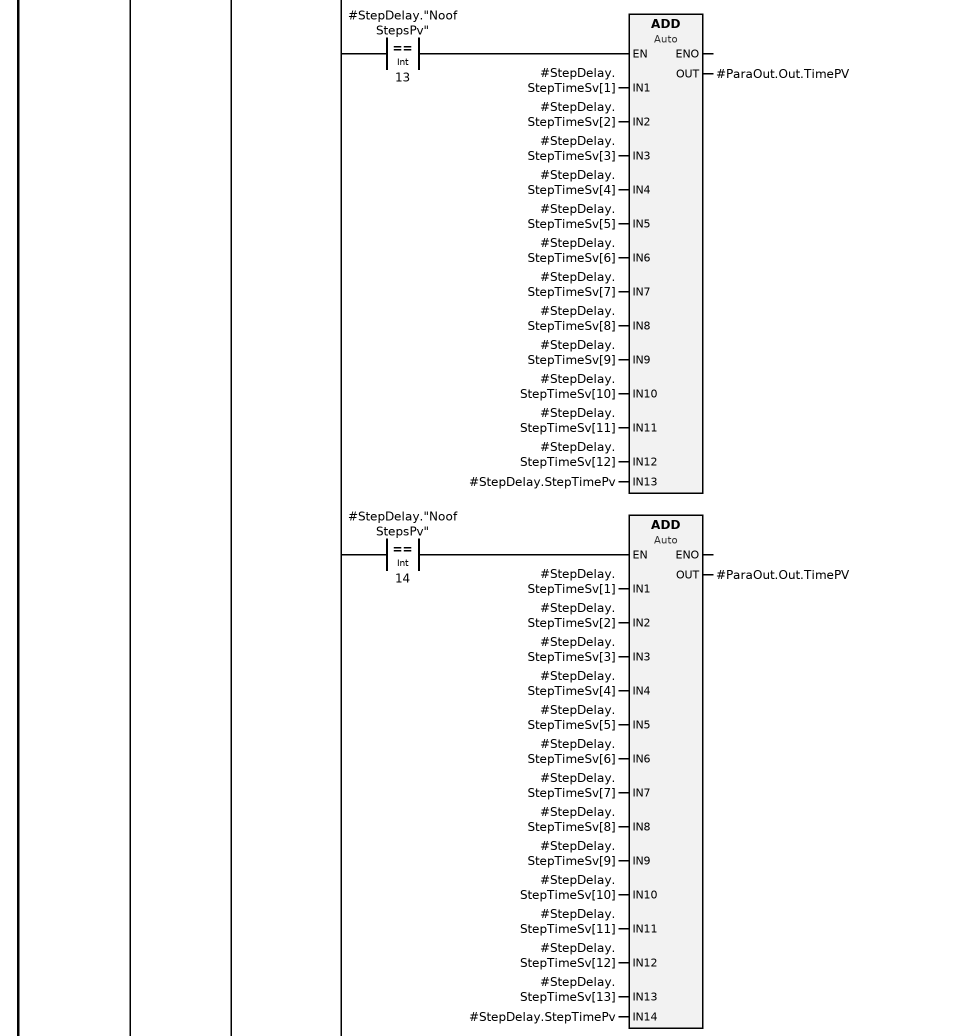
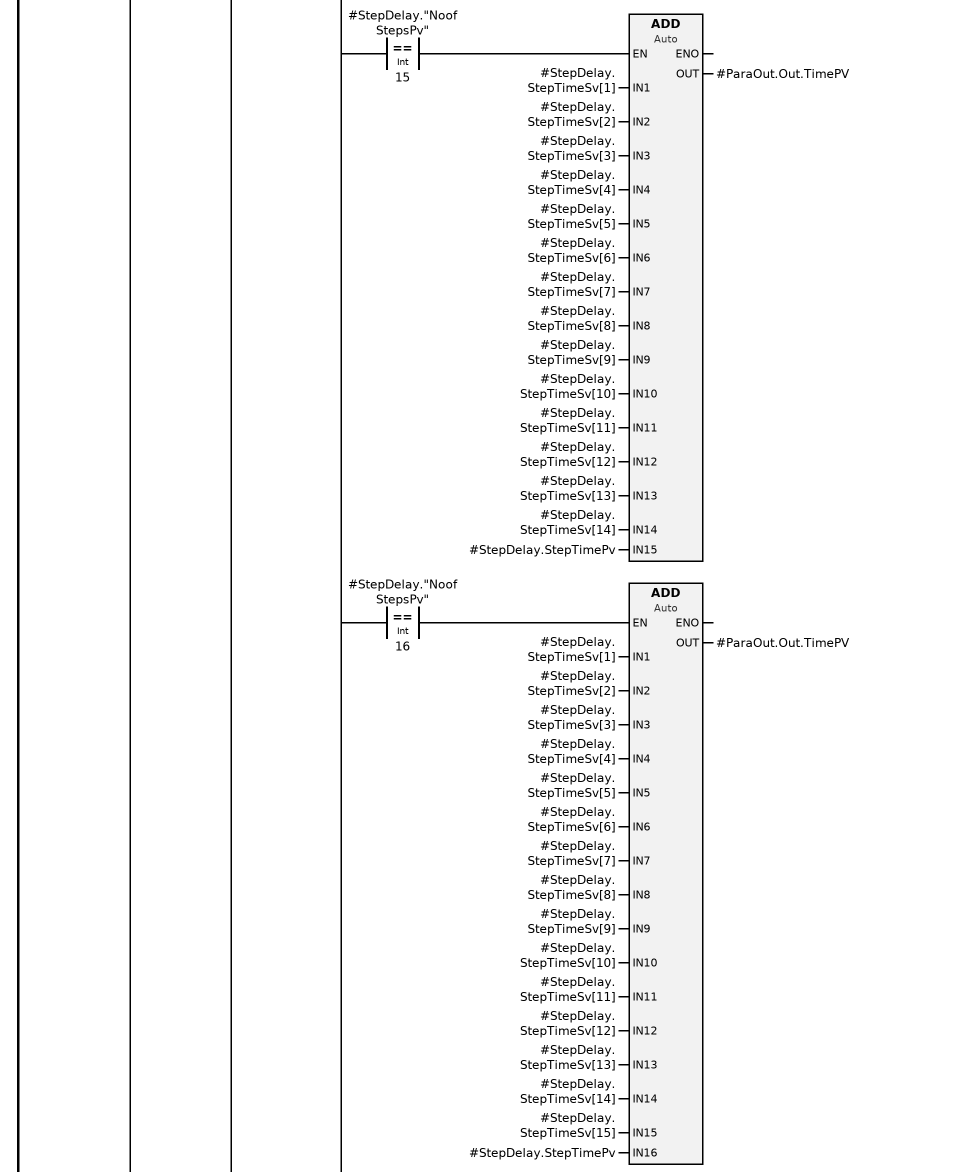
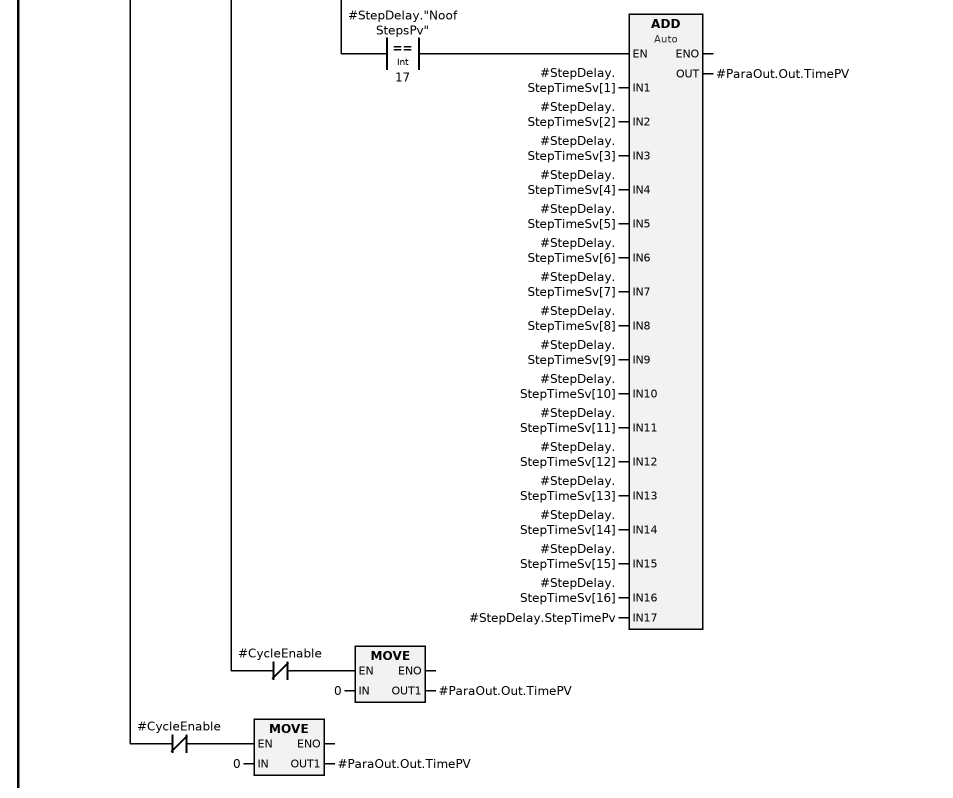
   RUNG wire#powerrail
      Contact( "AlwaysTRUE" )
      wire#w1
      { S7_Templates := "SrcType := DInt" } GE_Contact(in1 := #StepDelay.StepTimePv, in2 := 0)
      wire#w2
      { S7_Templates := "SrcType := Int" } LE_Contact(in1 := #ParaIn.PreciseEngineering.Loops, in2 := 20)
      wire#w3
      Add(in1 := #StepDelay.StepTimeSv[1], in2 := #StepDelay.StepTimeSv[2], in3 := #StepDelay.StepTimeSv[3], in4 := #StepDelay.StepTimeSv[4], in5 := #StepDelay.StepTimeSv[5], in6 := #StepDelay.StepTimeSv[6], in7 := #StepDelay.StepTimeSv[7], in8 := #StepDelay.StepTimeSv[8], in9 := #StepDelay.StepTimeSv[9], in10 := #StepDelay.StepTimeSv[10], in11 := #StepDelay.StepTimeSv[11], in12 := #StepDelay.StepTimeSv[12], in13 := #StepDelay.StepTimeSv[13], in14 := #StepDelay.StepTimeSv[14], in15 := #StepDelay.StepTimeSv[15], in16 := #StepDelay.StepTimeSv[16], in17 := #StepDelay.StepTimeSv[17], out => #ParaOut.Out.TimeSV)
   END_RUNG
   RUNG wire#w3
      Contact( #OverTemp )
      Add(in1 := #StepDelay.StepTimeSv[1], in2 := #StepDelay.StepTimeSv[2], in3 := #StepDelay.StepTimeSv[3], in4 := #StepDelay.StepTimeSv[4], in5 := #StepDelay.StepTimeSv[5], in6 := #StepDelay.StepTimeSv[6], in7 := #StepDelay.StepTimeSv[7], in8 := #StepDelay.StepTimeSv[8], in9 := #StepDelay.StepTimeSv[9], in10 := #StepDelay.StepTimeSv[10], in11 := #StepDelay.StepTimeSv[11], in12 := #StepDelay.StepTimeSv[12], in13 := #StepDelay.StepTimeSv[13], in14 := #StepDelay.StepTimeSv[14], in15 := #StepDelay.StepTimeSv[15], in16 := #StepDelay.StepTimeSv[16], in17 := #StepDelay.StepTimeSv[17], out => #ParaOut.Out.TimePV)
   END_RUNG
   RUNG wire#w2
      { S7_Templates := "SrcType := Int" } EQ_Contact(in1 := #ParaIn.PreciseEngineering.Loops, in2 := 5)
      I_Contact( #AlwaysTrue )
      wire#w4
      Add(in1 := #StepDelay.StepTimeSv[1], in2 := #StepDelay.StepTimeSv[2], in3 := #StepDelay.StepTimeSv[3], in4 := #StepDelay.StepTimeSv[4], in5 := #StepDelay.StepTimeSv[5], out => #ParaOut.Out.TimeSV)
   END_RUNG
   RUNG wire#w4
      Contact( #OverTemp )
      Add(in1 := #StepDelay.StepTimeSv[1], in2 := #StepDelay.StepTimeSv[2], in3 := #StepDelay.StepTimeSv[3], in4 := #StepDelay.StepTimeSv[4], in5 := #StepDelay.StepTimeSv[5], out => #ParaOut.Out.TimePV)
   END_RUNG
   RUNG wire#w2
      Contact( #CycleEnable )
      wire#w5
      { S7_Templates := "SrcType := Int" } EQ_Contact(in1 := #StepDelay."Noof StepsPv", in2 := 1)
      Move(in := #StepDelay.StepTimePv, out1 => #ParaOut.Out.TimePV)
   END_RUNG
   RUNG wire#w5
      { S7_Templates := "SrcType := Int" } EQ_Contact(in1 := #StepDelay."Noof StepsPv", in2 := 2)
      Add(in1 := #StepDelay.StepTimeSv[1], in2 := #StepDelay.StepTimePv, out => #ParaOut.Out.TimePV)
   END_RUNG
   RUNG wire#w5
      { S7_Templates := "SrcType := Int" } EQ_Contact(in1 := #StepDelay."Noof StepsPv", in2 := 3)
      Add(in1 := #StepDelay.StepTimeSv[1], in2 := #StepDelay.StepTimeSv[2], in3 := #StepDelay.StepTimePv, out => #ParaOut.Out.TimePV)
   END_RUNG
   RUNG wire#w5
      { S7_Templates := "SrcType := Int" } EQ_Contact(in1 := #StepDelay."Noof StepsPv", in2 := 4)
      Add(in1 := #StepDelay.StepTimeSv[1], in2 := #StepDelay.StepTimeSv[2], in3 := #StepDelay.StepTimeSv[3], in4 := #StepDelay.StepTimePv, out => #ParaOut.Out.TimePV)
   END_RUNG
   RUNG wire#w5
      { S7_Templates := "SrcType := Int" } EQ_Contact(in1 := #StepDelay."Noof StepsPv", in2 := 5)
      Add(in1 := #StepDelay.StepTimeSv[1], in2 := #StepDelay.StepTimeSv[2], in3 := #StepDelay.StepTimeSv[3], in4 := #StepDelay.StepTimeSv[4], in5 := #StepDelay.StepTimePv, out => #ParaOut.Out.TimePV)
   END_RUNG
   RUNG wire#w5
      { S7_Templates := "SrcType := Int" } EQ_Contact(in1 := #StepDelay."Noof StepsPv", in2 := 6)
      Add(in1 := #StepDelay.StepTimeSv[1], in2 := #StepDelay.StepTimeSv[2], in3 := #StepDelay.StepTimeSv[3], in4 := #StepDelay.StepTimeSv[4], in5 := #StepDelay.StepTimeSv[5], in6 := #StepDelay.StepTimePv, out => #ParaOut.Out.TimePV)
   END_RUNG
   RUNG wire#w5
      { S7_Templates := "SrcType := Int" } EQ_Contact(in1 := #StepDelay."Noof StepsPv", in2 := 7)
      Add(in1 := #StepDelay.StepTimeSv[1], in2 := #StepDelay.StepTimeSv[2], in3 := #StepDelay.StepTimeSv[3], in4 := #StepDelay.StepTimeSv[4], in5 := #StepDelay.StepTimeSv[5], in6 := #StepDelay.StepTimeSv[6], in7 := #StepDelay.StepTimePv, out => #ParaOut.Out.TimePV)
   END_RUNG
   RUNG wire#w5
      { S7_Templates := "SrcType := Int" } EQ_Contact(in1 := #StepDelay."Noof StepsPv", in2 := 8)
      Add(in1 := #StepDelay.StepTimeSv[1], in2 := #StepDelay.StepTimeSv[2], in3 := #StepDelay.StepTimeSv[3], in4 := #StepDelay.StepTimeSv[4], in5 := #StepDelay.StepTimeSv[5], in6 := #StepDelay.StepTimeSv[6], in7 := #StepDelay.StepTimeSv[7], in8 := #StepDelay.StepTimePv, out => #ParaOut.Out.TimePV)
   END_RUNG
   RUNG wire#w5
      { S7_Templates := "SrcType := Int" } EQ_Contact(in1 := #StepDelay."Noof StepsPv", in2 := 9)
      Add(in1 := #StepDelay.StepTimeSv[1], in2 := #StepDelay.StepTimeSv[2], in3 := #StepDelay.StepTimeSv[3], in4 := #StepDelay.StepTimeSv[4], in5 := #StepDelay.StepTimeSv[5], in6 := #StepDelay.StepTimeSv[6], in7 := #StepDelay.StepTimeSv[7], in8 := #StepDelay.StepTimeSv[8], in9 := #StepDelay.StepTimePv, out => #ParaOut.Out.TimePV)
   END_RUNG
   RUNG wire#w5
      { S7_Templates := "SrcType := Int" } EQ_Contact(in1 := #StepDelay."Noof StepsPv", in2 := 10)
      Add(in1 := #StepDelay.StepTimeSv[1], in2 := #StepDelay.StepTimeSv[2], in3 := #StepDelay.StepTimeSv[3], in4 := #StepDelay.StepTimeSv[4], in5 := #StepDelay.StepTimeSv[5], in6 := #StepDelay.StepTimeSv[6], in7 := #StepDelay.StepTimeSv[7], in8 := #StepDelay.StepTimeSv[8], in9 := #StepDelay.StepTimeSv[9], in10 := #StepDelay.StepTimePv, out => #ParaOut.Out.TimePV)
   END_RUNG
   RUNG wire#w5
      { S7_Templates := "SrcType := Int" } EQ_Contact(in1 := #StepDelay."Noof StepsPv", in2 := 11)
      Add(in1 := #StepDelay.StepTimeSv[1], in2 := #StepDelay.StepTimeSv[2], in3 := #StepDelay.StepTimeSv[3], in4 := #StepDelay.StepTimeSv[4], in5 := #StepDelay.StepTimeSv[5], in6 := #StepDelay.StepTimeSv[6], in7 := #StepDelay.StepTimeSv[7], in8 := #StepDelay.StepTimeSv[8], in9 := #StepDelay.StepTimeSv[9], in10 := #StepDelay.StepTimeSv[10], in11 := #StepDelay.StepTimePv, out => #ParaOut.Out.TimePV)
   END_RUNG
   RUNG wire#w5
      { S7_Templates := "SrcType := Int" } EQ_Contact(in1 := #StepDelay."Noof StepsPv", in2 := 12)
      Add(in1 := #StepDelay.StepTimeSv[1], in2 := #StepDelay.StepTimeSv[2], in3 := #StepDelay.StepTimeSv[3], in4 := #StepDelay.StepTimeSv[4], in5 := #StepDelay.StepTimeSv[5], in6 := #StepDelay.StepTimeSv[6], in7 := #StepDelay.StepTimeSv[7], in8 := #StepDelay.StepTimeSv[8], in9 := #StepDelay.StepTimeSv[9], in10 := #StepDelay.StepTimeSv[10], in11 := #StepDelay.StepTimeSv[11], in12 := #StepDelay.StepTimePv, out => #ParaOut.Out.TimePV)
   END_RUNG
   RUNG wire#w5
      { S7_Templates := "SrcType := Int" } EQ_Contact(in1 := #StepDelay."Noof StepsPv", in2 := 13)
      Add(in1 := #StepDelay.StepTimeSv[1], in2 := #StepDelay.StepTimeSv[2], in3 := #StepDelay.StepTimeSv[3], in4 := #StepDelay.StepTimeSv[4], in5 := #StepDelay.StepTimeSv[5], in6 := #StepDelay.StepTimeSv[6], in7 := #StepDelay.StepTimeSv[7], in8 := #StepDelay.StepTimeSv[8], in9 := #StepDelay.StepTimeSv[9], in10 := #StepDelay.StepTimeSv[10], in11 := #StepDelay.StepTimeSv[11], in12 := #StepDelay.StepTimeSv[12], in13 := #StepDelay.StepTimePv, out => #ParaOut.Out.TimePV)
   END_RUNG
   RUNG wire#w5
      { S7_Templates := "SrcType := Int" } EQ_Contact(in1 := #StepDelay."Noof StepsPv", in2 := 14)
      Add(in1 := #StepDelay.StepTimeSv[1], in2 := #StepDelay.StepTimeSv[2], in3 := #StepDelay.StepTimeSv[3], in4 := #StepDelay.StepTimeSv[4], in5 := #StepDelay.StepTimeSv[5], in6 := #StepDelay.StepTimeSv[6], in7 := #StepDelay.StepTimeSv[7], in8 := #StepDelay.StepTimeSv[8], in9 := #StepDelay.StepTimeSv[9], in10 := #StepDelay.StepTimeSv[10], in11 := #StepDelay.StepTimeSv[11], in12 := #StepDelay.StepTimeSv[12], in13 := #StepDelay.StepTimeSv[13], in14 := #StepDelay.StepTimePv, out => #ParaOut.Out.TimePV)
   END_RUNG
   RUNG wire#w5
      { S7_Templates := "SrcType := Int" } EQ_Contact(in1 := #StepDelay."Noof StepsPv", in2 := 15)
      Add(in1 := #StepDelay.StepTimeSv[1], in2 := #StepDelay.StepTimeSv[2], in3 := #StepDelay.StepTimeSv[3], in4 := #StepDelay.StepTimeSv[4], in5 := #StepDelay.StepTimeSv[5], in6 := #StepDelay.StepTimeSv[6], in7 := #StepDelay.StepTimeSv[7], in8 := #StepDelay.StepTimeSv[8], in9 := #StepDelay.StepTimeSv[9], in10 := #StepDelay.StepTimeSv[10], in11 := #StepDelay.StepTimeSv[11], in12 := #StepDelay.StepTimeSv[12], in13 := #StepDelay.StepTimeSv[13], in14 := #StepDelay.StepTimeSv[14], in15 := #StepDelay.StepTimePv, out => #ParaOut.Out.TimePV)
   END_RUNG
   RUNG wire#w5
      { S7_Templates := "SrcType := Int" } EQ_Contact(in1 := #StepDelay."Noof StepsPv", in2 := 16)
      Add(in1 := #StepDelay.StepTimeSv[1], in2 := #StepDelay.StepTimeSv[2], in3 := #StepDelay.StepTimeSv[3], in4 := #StepDelay.StepTimeSv[4], in5 := #StepDelay.StepTimeSv[5], in6 := #StepDelay.StepTimeSv[6], in7 := #StepDelay.StepTimeSv[7], in8 := #StepDelay.StepTimeSv[8], in9 := #StepDelay.StepTimeSv[9], in10 := #StepDelay.StepTimeSv[10], in11 := #StepDelay.StepTimeSv[11], in12 := #StepDelay.StepTimeSv[12], in13 := #StepDelay.StepTimeSv[13], in14 := #StepDelay.StepTimeSv[14], in15 := #StepDelay.StepTimeSv[15], in16 := #StepDelay.StepTimePv, out => #ParaOut.Out.TimePV)
   END_RUNG
   RUNG wire#w5
      { S7_Templates := "SrcType := Int" } EQ_Contact(in1 := #StepDelay."Noof StepsPv", in2 := 17)
      Add(in1 := #StepDelay.StepTimeSv[1], in2 := #StepDelay.StepTimeSv[2], in3 := #StepDelay.StepTimeSv[3], in4 := #StepDelay.StepTimeSv[4], in5 := #StepDelay.StepTimeSv[5], in6 := #StepDelay.StepTimeSv[6], in7 := #StepDelay.StepTimeSv[7], in8 := #StepDelay.StepTimeSv[8], in9 := #StepDelay.StepTimeSv[9], in10 := #StepDelay.StepTimeSv[10], in11 := #StepDelay.StepTimeSv[11], in12 := #StepDelay.StepTimeSv[12], in13 := #StepDelay.StepTimeSv[13], in14 := #StepDelay.StepTimeSv[14], in15 := #StepDelay.StepTimeSv[15], in16 := #StepDelay.StepTimeSv[16], in17 := #StepDelay.StepTimePv, out => #ParaOut.Out.TimePV)
   END_RUNG
   RUNG wire#w2
      I_Contact( #CycleEnable )
      Move(in := 0, out1 => #ParaOut.Out.TimePV)
   END_RUNG
   RUNG wire#w1
      I_Contact( #CycleEnable )
      Move(in := 0, out1 => #ParaOut.Out.TimePV)
   END_RUNG
   // the same network as SCL:
   #_w1 := "AlwaysTRUE" AND (#StepDelay.StepTimePv >= 0);
   #_w2 := #_w1 AND (#ParaIn.PreciseEngineering.Loops <= 20);
   IF #_w2 THEN
       #ParaOut.Out.TimeSV := #StepDelay.StepTimeSv[1] + #StepDelay.StepTimeSv[2] + #StepDelay.StepTimeSv[3] + #StepDelay.StepTimeSv[4] + #StepDelay.StepTimeSv[5] + #StepDelay.StepTimeSv[6] + #StepDelay.StepTimeSv[7] + #StepDelay.StepTimeSv[8] + #StepDelay.StepTimeSv[9] + #StepDelay.StepTimeSv[10] + #StepDelay.StepTimeSv[11] + #StepDelay.StepTimeSv[12] + #StepDelay.StepTimeSv[13] + #StepDelay.StepTimeSv[14] + #StepDelay.StepTimeSv[15] + #StepDelay.StepTimeSv[16] + #StepDelay.StepTimeSv[17];
   END_IF;
   IF #_w2 AND #OverTemp THEN
       #ParaOut.Out.TimePV := #StepDelay.StepTimeSv[1] + #StepDelay.StepTimeSv[2] + #StepDelay.StepTimeSv[3] + #StepDelay.StepTimeSv[4] + #StepDelay.StepTimeSv[5] + #StepDelay.StepTimeSv[6] + #StepDelay.StepTimeSv[7] + #StepDelay.StepTimeSv[8] + #StepDelay.StepTimeSv[9] + #StepDelay.StepTimeSv[10] + #StepDelay.StepTimeSv[11] + #StepDelay.StepTimeSv[12] + #StepDelay.StepTimeSv[13] + #StepDelay.StepTimeSv[14] + #StepDelay.StepTimeSv[15] + #StepDelay.StepTimeSv[16] + #StepDelay.StepTimeSv[17];
   END_IF;
   #_w3 := #_w1 AND (#ParaIn.PreciseEngineering.Loops = 5) AND NOT #AlwaysTrue;
   IF #_w3 THEN
       #ParaOut.Out.TimeSV := #StepDelay.StepTimeSv[1] + #StepDelay.StepTimeSv[2] + #StepDelay.StepTimeSv[3] + #StepDelay.StepTimeSv[4] + #StepDelay.StepTimeSv[5];
   END_IF;
   IF #_w3 AND #OverTemp THEN
       #ParaOut.Out.TimePV := #StepDelay.StepTimeSv[1] + #StepDelay.StepTimeSv[2] + #StepDelay.StepTimeSv[3] + #StepDelay.StepTimeSv[4] + #StepDelay.StepTimeSv[5];
   END_IF;
   #_w4 := #_w1 AND #CycleEnable;
   IF #_w4 AND (#StepDelay."Noof StepsPv" = 1) THEN #ParaOut.Out.TimePV := #StepDelay.StepTimePv; END_IF;
   IF #_w4 AND (#StepDelay."Noof StepsPv" = 2) THEN
       #ParaOut.Out.TimePV := #StepDelay.StepTimeSv[1] + #StepDelay.StepTimePv;
   END_IF;
   IF #_w4 AND (#StepDelay."Noof StepsPv" = 3) THEN
       #ParaOut.Out.TimePV := #StepDelay.StepTimeSv[1] + #StepDelay.StepTimeSv[2] + #StepDelay.StepTimePv;
   END_IF;
   IF #_w4 AND (#StepDelay."Noof StepsPv" = 4) THEN
       #ParaOut.Out.TimePV := #StepDelay.StepTimeSv[1] + #StepDelay.StepTimeSv[2] + #StepDelay.StepTimeSv[3] + #StepDelay.StepTimePv;
   END_IF;
   IF #_w4 AND (#StepDelay."Noof StepsPv" = 5) THEN
       #ParaOut.Out.TimePV := #StepDelay.StepTimeSv[1] + #StepDelay.StepTimeSv[2] + #StepDelay.StepTimeSv[3] + #StepDelay.StepTimeSv[4] + #StepDelay.StepTimePv;
   END_IF;
   IF #_w4 AND (#StepDelay."Noof StepsPv" = 6) THEN
       #ParaOut.Out.TimePV := #StepDelay.StepTimeSv[1] + #StepDelay.StepTimeSv[2] + #StepDelay.StepTimeSv[3] + #StepDelay.StepTimeSv[4] + #StepDelay.StepTimeSv[5] + #StepDelay.StepTimePv;
   END_IF;
   IF #_w4 AND (#StepDelay."Noof StepsPv" = 7) THEN
       #ParaOut.Out.TimePV := #StepDelay.StepTimeSv[1] + #StepDelay.StepTimeSv[2] + #StepDelay.StepTimeSv[3] + #StepDelay.StepTimeSv[4] + #StepDelay.StepTimeSv[5] + #StepDelay.StepTimeSv[6] + #StepDelay.StepTimePv;
   END_IF;
   IF #_w4 AND (#StepDelay."Noof StepsPv" = 8) THEN
       #ParaOut.Out.TimePV := #StepDelay.StepTimeSv[1] + #StepDelay.StepTimeSv[2] + #StepDelay.StepTimeSv[3] + #StepDelay.StepTimeSv[4] + #StepDelay.StepTimeSv[5] + #StepDelay.StepTimeSv[6] + #StepDelay.StepTimeSv[7] + #StepDelay.StepTimePv;
   END_IF;
   IF #_w4 AND (#StepDelay."Noof StepsPv" = 9) THEN
       #ParaOut.Out.TimePV := #StepDelay.StepTimeSv[1] + #StepDelay.StepTimeSv[2] + #StepDelay.StepTimeSv[3] + #StepDelay.StepTimeSv[4] + #StepDelay.StepTimeSv[5] + #StepDelay.StepTimeSv[6] + #StepDelay.StepTimeSv[7] + #StepDelay.StepTimeSv[8] + #StepDelay.StepTimePv;
   END_IF;
   IF #_w4 AND (#StepDelay."Noof StepsPv" = 10) THEN
       #ParaOut.Out.TimePV := #StepDelay.StepTimeSv[1] + #StepDelay.StepTimeSv[2] + #StepDelay.StepTimeSv[3] + #StepDelay.StepTimeSv[4] + #StepDelay.StepTimeSv[5] + #StepDelay.StepTimeSv[6] + #StepDelay.StepTimeSv[7] + #StepDelay.StepTimeSv[8] + #StepDelay.StepTimeSv[9] + #StepDelay.StepTimePv;
   END_IF;
   IF #_w4 AND (#StepDelay."Noof StepsPv" = 11) THEN
       #ParaOut.Out.TimePV := #StepDelay.StepTimeSv[1] + #StepDelay.StepTimeSv[2] + #StepDelay.StepTimeSv[3] + #StepDelay.StepTimeSv[4] + #StepDelay.StepTimeSv[5] + #StepDelay.StepTimeSv[6] + #StepDelay.StepTimeSv[7] + #StepDelay.StepTimeSv[8] + #StepDelay.StepTimeSv[9] + #StepDelay.StepTimeSv[10] + #StepDelay.StepTimePv;
   END_IF;
   IF #_w4 AND (#StepDelay."Noof StepsPv" = 12) THEN
       #ParaOut.Out.TimePV := #StepDelay.StepTimeSv[1] + #StepDelay.StepTimeSv[2] + #StepDelay.StepTimeSv[3] + #StepDelay.StepTimeSv[4] + #StepDelay.StepTimeSv[5] + #StepDelay.StepTimeSv[6] + #StepDelay.StepTimeSv[7] + #StepDelay.StepTimeSv[8] + #StepDelay.StepTimeSv[9] + #StepDelay.StepTimeSv[10] + #StepDelay.StepTimeSv[11] + #StepDelay.StepTimePv;
   END_IF;
   IF #_w4 AND (#StepDelay."Noof StepsPv" = 13) THEN
       #ParaOut.Out.TimePV := #StepDelay.StepTimeSv[1] + #StepDelay.StepTimeSv[2] + #StepDelay.StepTimeSv[3] + #StepDelay.StepTimeSv[4] + #StepDelay.StepTimeSv[5] + #StepDelay.StepTimeSv[6] + #StepDelay.StepTimeSv[7] + #StepDelay.StepTimeSv[8] + #StepDelay.StepTimeSv[9] + #StepDelay.StepTimeSv[10] + #StepDelay.StepTimeSv[11] + #StepDelay.StepTimeSv[12] + #StepDelay.StepTimePv;
   END_IF;
   IF #_w4 AND (#StepDelay."Noof StepsPv" = 14) THEN
       #ParaOut.Out.TimePV := #StepDelay.StepTimeSv[1] + #StepDelay.StepTimeSv[2] + #StepDelay.StepTimeSv[3] + #StepDelay.StepTimeSv[4] + #StepDelay.StepTimeSv[5] + #StepDelay.StepTimeSv[6] + #StepDelay.StepTimeSv[7] + #StepDelay.StepTimeSv[8] + #StepDelay.StepTimeSv[9] + #StepDelay.StepTimeSv[10] + #StepDelay.StepTimeSv[11] + #StepDelay.StepTimeSv[12] + #StepDelay.StepTimeSv[13] + #StepDelay.StepTimePv;
   END_IF;
   IF #_w4 AND (#StepDelay."Noof StepsPv" = 15) THEN
       #ParaOut.Out.TimePV := #StepDelay.StepTimeSv[1] + #StepDelay.StepTimeSv[2] + #StepDelay.StepTimeSv[3] + #StepDelay.StepTimeSv[4] + #StepDelay.StepTimeSv[5] + #StepDelay.StepTimeSv[6] + #StepDelay.StepTimeSv[7] + #StepDelay.StepTimeSv[8] + #StepDelay.StepTimeSv[9] + #StepDelay.StepTimeSv[10] + #StepDelay.StepTimeSv[11] + #StepDelay.StepTimeSv[12] + #StepDelay.StepTimeSv[13] + #StepDelay.StepTimeSv[14] + #StepDelay.StepTimePv;
   END_IF;
   IF #_w4 AND (#StepDelay."Noof StepsPv" = 16) THEN
       #ParaOut.Out.TimePV := #StepDelay.StepTimeSv[1] + #StepDelay.StepTimeSv[2] + #StepDelay.StepTimeSv[3] + #StepDelay.StepTimeSv[4] + #StepDelay.StepTimeSv[5] + #StepDelay.StepTimeSv[6] + #StepDelay.StepTimeSv[7] + #StepDelay.StepTimeSv[8] + #StepDelay.StepTimeSv[9] + #StepDelay.StepTimeSv[10] + #StepDelay.StepTimeSv[11] + #StepDelay.StepTimeSv[12] + #StepDelay.StepTimeSv[13] + #StepDelay.StepTimeSv[14] + #StepDelay.StepTimeSv[15] + #StepDelay.StepTimePv;
   END_IF;
   IF #_w4 AND (#StepDelay."Noof StepsPv" = 17) THEN
       #ParaOut.Out.TimePV := #StepDelay.StepTimeSv[1] + #StepDelay.StepTimeSv[2] + #StepDelay.StepTimeSv[3] + #StepDelay.StepTimeSv[4] + #StepDelay.StepTimeSv[5] + #StepDelay.StepTimeSv[6] + #StepDelay.StepTimeSv[7] + #StepDelay.StepTimeSv[8] + #StepDelay.StepTimeSv[9] + #StepDelay.StepTimeSv[10] + #StepDelay.StepTimeSv[11] + #StepDelay.StepTimeSv[12] + #StepDelay.StepTimeSv[13] + #StepDelay.StepTimeSv[14] + #StepDelay.StepTimeSv[15] + #StepDelay.StepTimeSv[16] + #StepDelay.StepTimePv;
   END_IF;
   IF #_w1 AND NOT #CycleEnable THEN #ParaOut.Out.TimePV := 0; END_IF;
   IF "AlwaysTRUE" AND NOT #CycleEnable THEN #ParaOut.Out.TimePV := 0; END_IF;
END_REGION

REGION Network 12: #StepDelay
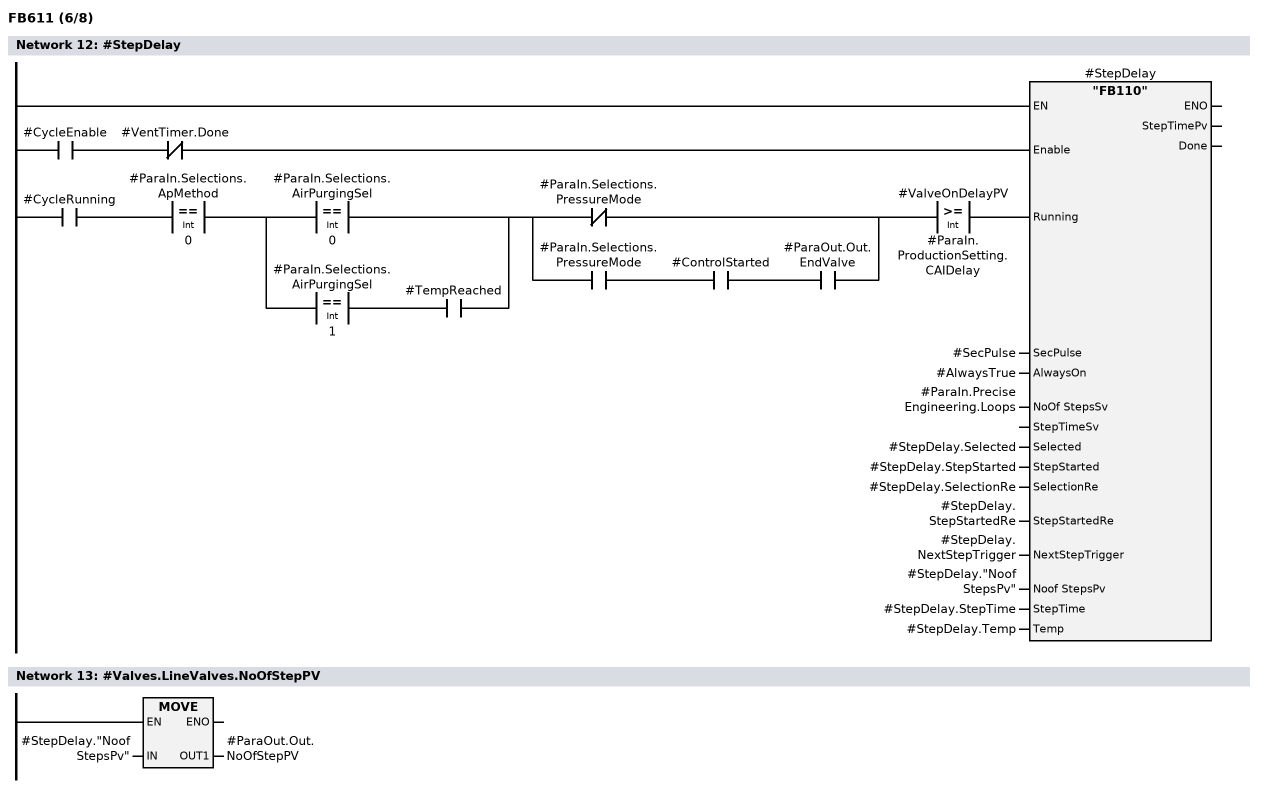
   RUNG wire#powerrail
      #StepDelay(Enable := wire#w1, Running := wire#w5, SecPulse := #SecPulse, AlwaysOn := #AlwaysTrue, "NoOf StepsSv" := #ParaIn.PreciseEngineering.Loops, StepTimeSv :=, Selected := #StepDelay.Selected, StepStarted := #StepDelay.StepStarted, SelectionRe := #StepDelay.SelectionRe, StepStartedRe := #StepDelay.StepStartedRe, NextStepTrigger := #StepDelay.NextStepTrigger, "Noof StepsPv" := #StepDelay."Noof StepsPv", StepTime := #StepDelay.StepTime, Temp := #StepDelay.Temp, StepTimePv =>, Done =>)
   END_RUNG
   RUNG wire#powerrail
      Contact( #CycleEnable )
      I_Contact( #VentTimer.Done )
   END_RUNG wire#w1
   RUNG wire#powerrail
      Contact( #CycleRunning )
      { S7_Templates := "SrcType := Int" } EQ_Contact(in1 := #ParaIn.Selections.ApMethod, in2 := 0)
      wire#w2
      { S7_Templates := "SrcType := Int" } EQ_Contact(in1 := #ParaIn.Selections.AirPurgingSel, in2 := 0)
      wire#w3
      I_Contact( #ParaIn.Selections.PressureMode )
      wire#w4
      { S7_Templates := "SrcType := Int" } GE_Contact(in1 := #ValveOnDelayPV, in2 := #ParaIn.ProductionSetting.CAIDelay)
   END_RUNG wire#w5
   RUNG wire#w2
      { S7_Templates := "SrcType := Int" } EQ_Contact(in1 := #ParaIn.Selections.AirPurgingSel, in2 := 1)
      Contact( #TempReached )
   END_RUNG wire#w3
   RUNG wire#w3
      Contact( #ParaIn.Selections.PressureMode )
      Contact( #ControlStarted )
      Contact( #ParaOut.Out.EndValve )
   END_RUNG wire#w4
   // the same network as SCL:
   #StepDelay(Enable := #CycleEnable AND NOT #VentTimer.Done,   // "FB110"
              Running := #CycleRunning AND (#ParaIn.Selections.ApMethod = 0) AND ((#ParaIn.Selections.AirPurgingSel = 0) OR ((#ParaIn.Selections.AirPurgingSel = 1) AND #TempReached)) AND (NOT #ParaIn.Selections.PressureMode OR (#ParaIn.Selections.PressureMode AND #ControlStarted AND #ParaOut.Out.EndValve)) AND (#ValveOnDelayPV >= #ParaIn.ProductionSetting.CAIDelay),
              SecPulse := #SecPulse,
              AlwaysOn := #AlwaysTrue,
              "NoOf StepsSv" := #ParaIn.PreciseEngineering.Loops,
              Selected := #StepDelay.Selected,
              StepStarted := #StepDelay.StepStarted,
              SelectionRe := #StepDelay.SelectionRe,
              StepStartedRe := #StepDelay.StepStartedRe,
              NextStepTrigger := #StepDelay.NextStepTrigger,
              "Noof StepsPv" := #StepDelay."Noof StepsPv",
              StepTime := #StepDelay.StepTime,
              Temp := #StepDelay.Temp);
END_REGION

REGION Network 13: #Valves.LineValves.NoOfStepPV
   RUNG wire#powerrail
      Move(in := #StepDelay."Noof StepsPv", out1 => #ParaOut.Out.NoOfStepPV)
   END_RUNG
   // the same network as SCL:
   #ParaOut.Out.NoOfStepPV := #StepDelay."Noof StepsPv";
END_REGION

REGION Network 14: Loop Outputs
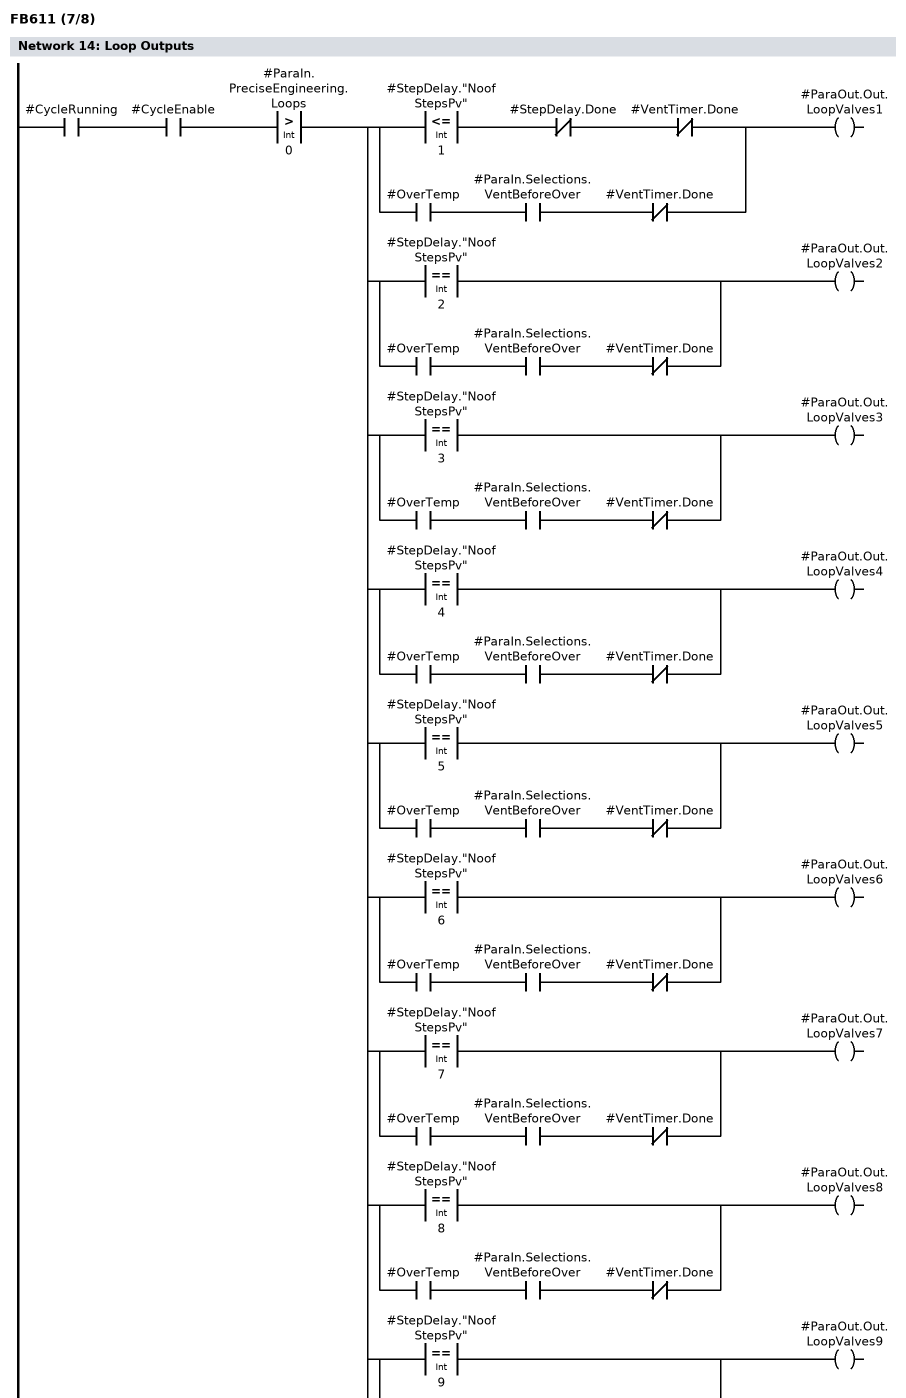
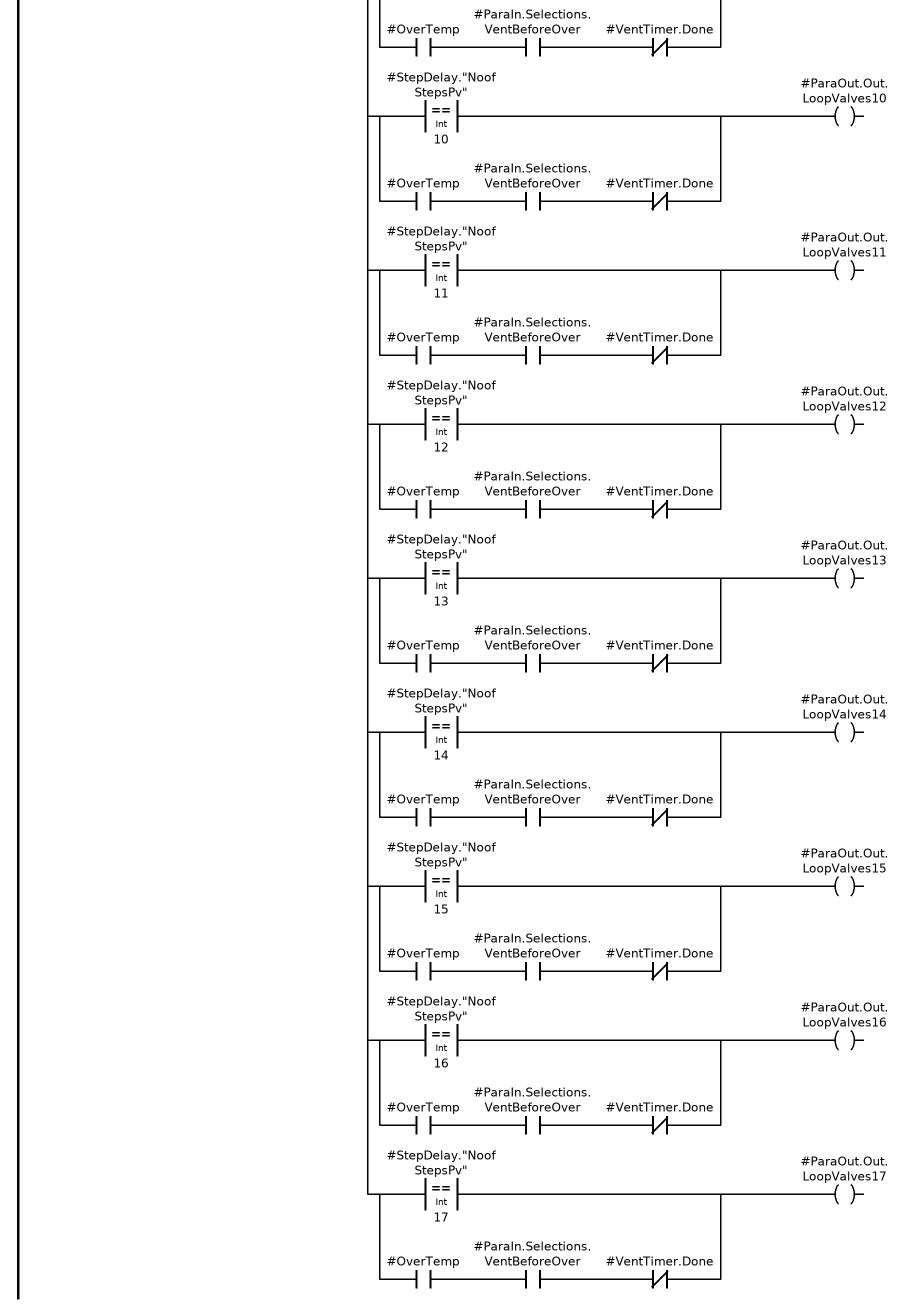
   RUNG wire#powerrail
      Contact( #CycleRunning )
      Contact( #CycleEnable )
      { S7_Templates := "SrcType := Int" } GT_Contact(in1 := #ParaIn.PreciseEngineering.Loops, in2 := 0)
      wire#w1
      { S7_Templates := "SrcType := Int" } LE_Contact(in1 := #StepDelay."Noof StepsPv", in2 := 1)
      I_Contact( #StepDelay.Done )
      I_Contact( #VentTimer.Done )
      wire#w2
      Coil( #ParaOut.Out.LoopValves1 )
   END_RUNG
   RUNG wire#w1
      Contact( #OverTemp )
      Contact( #ParaIn.Selections.VentBeforeOver )
      I_Contact( #VentTimer.Done )
   END_RUNG wire#w2
   RUNG wire#w1
      { S7_Templates := "SrcType := Int" } EQ_Contact(in1 := #StepDelay."Noof StepsPv", in2 := 2)
      wire#w3
      Coil( #ParaOut.Out.LoopValves2 )
   END_RUNG
   RUNG wire#w1
      Contact( #OverTemp )
      Contact( #ParaIn.Selections.VentBeforeOver )
      I_Contact( #VentTimer.Done )
   END_RUNG wire#w3
   RUNG wire#w1
      { S7_Templates := "SrcType := Int" } EQ_Contact(in1 := #StepDelay."Noof StepsPv", in2 := 3)
      wire#w4
      Coil( #ParaOut.Out.LoopValves3 )
   END_RUNG
   RUNG wire#w1
      Contact( #OverTemp )
      Contact( #ParaIn.Selections.VentBeforeOver )
      I_Contact( #VentTimer.Done )
   END_RUNG wire#w4
   RUNG wire#w1
      { S7_Templates := "SrcType := Int" } EQ_Contact(in1 := #StepDelay."Noof StepsPv", in2 := 4)
      wire#w5
      Coil( #ParaOut.Out.LoopValves4 )
   END_RUNG
   RUNG wire#w1
      Contact( #OverTemp )
      Contact( #ParaIn.Selections.VentBeforeOver )
      I_Contact( #VentTimer.Done )
   END_RUNG wire#w5
   RUNG wire#w1
      { S7_Templates := "SrcType := Int" } EQ_Contact(in1 := #StepDelay."Noof StepsPv", in2 := 5)
      wire#w6
      Coil( #ParaOut.Out.LoopValves5 )
   END_RUNG
   RUNG wire#w1
      Contact( #OverTemp )
      Contact( #ParaIn.Selections.VentBeforeOver )
      I_Contact( #VentTimer.Done )
   END_RUNG wire#w6
   RUNG wire#w1
      { S7_Templates := "SrcType := Int" } EQ_Contact(in1 := #StepDelay."Noof StepsPv", in2 := 6)
      wire#w7
      Coil( #ParaOut.Out.LoopValves6 )
   END_RUNG
   RUNG wire#w1
      Contact( #OverTemp )
      Contact( #ParaIn.Selections.VentBeforeOver )
      I_Contact( #VentTimer.Done )
   END_RUNG wire#w7
   RUNG wire#w1
      { S7_Templates := "SrcType := Int" } EQ_Contact(in1 := #StepDelay."Noof StepsPv", in2 := 7)
      wire#w8
      Coil( #ParaOut.Out.LoopValves7 )
   END_RUNG
   RUNG wire#w1
      Contact( #OverTemp )
      Contact( #ParaIn.Selections.VentBeforeOver )
      I_Contact( #VentTimer.Done )
   END_RUNG wire#w8
   RUNG wire#w1
      { S7_Templates := "SrcType := Int" } EQ_Contact(in1 := #StepDelay."Noof StepsPv", in2 := 8)
      wire#w9
      Coil( #ParaOut.Out.LoopValves8 )
   END_RUNG
   RUNG wire#w1
      Contact( #OverTemp )
      Contact( #ParaIn.Selections.VentBeforeOver )
      I_Contact( #VentTimer.Done )
   END_RUNG wire#w9
   RUNG wire#w1
      { S7_Templates := "SrcType := Int" } EQ_Contact(in1 := #StepDelay."Noof StepsPv", in2 := 9)
      wire#w10
      Coil( #ParaOut.Out.LoopValves9 )
   END_RUNG
   RUNG wire#w1
      Contact( #OverTemp )
      Contact( #ParaIn.Selections.VentBeforeOver )
      I_Contact( #VentTimer.Done )
   END_RUNG wire#w10
   RUNG wire#w1
      { S7_Templates := "SrcType := Int" } EQ_Contact(in1 := #StepDelay."Noof StepsPv", in2 := 10)
      wire#w11
      Coil( #ParaOut.Out.LoopValves10 )
   END_RUNG
   RUNG wire#w1
      Contact( #OverTemp )
      Contact( #ParaIn.Selections.VentBeforeOver )
      I_Contact( #VentTimer.Done )
   END_RUNG wire#w11
   RUNG wire#w1
      { S7_Templates := "SrcType := Int" } EQ_Contact(in1 := #StepDelay."Noof StepsPv", in2 := 11)
      wire#w12
      Coil( #ParaOut.Out.LoopValves11 )
   END_RUNG
   RUNG wire#w1
      Contact( #OverTemp )
      Contact( #ParaIn.Selections.VentBeforeOver )
      I_Contact( #VentTimer.Done )
   END_RUNG wire#w12
   RUNG wire#w1
      { S7_Templates := "SrcType := Int" } EQ_Contact(in1 := #StepDelay."Noof StepsPv", in2 := 12)
      wire#w13
      Coil( #ParaOut.Out.LoopValves12 )
   END_RUNG
   RUNG wire#w1
      Contact( #OverTemp )
      Contact( #ParaIn.Selections.VentBeforeOver )
      I_Contact( #VentTimer.Done )
   END_RUNG wire#w13
   RUNG wire#w1
      { S7_Templates := "SrcType := Int" } EQ_Contact(in1 := #StepDelay."Noof StepsPv", in2 := 13)
      wire#w14
      Coil( #ParaOut.Out.LoopValves13 )
   END_RUNG
   RUNG wire#w1
      Contact( #OverTemp )
      Contact( #ParaIn.Selections.VentBeforeOver )
      I_Contact( #VentTimer.Done )
   END_RUNG wire#w14
   RUNG wire#w1
      { S7_Templates := "SrcType := Int" } EQ_Contact(in1 := #StepDelay."Noof StepsPv", in2 := 14)
      wire#w15
      Coil( #ParaOut.Out.LoopValves14 )
   END_RUNG
   RUNG wire#w1
      Contact( #OverTemp )
      Contact( #ParaIn.Selections.VentBeforeOver )
      I_Contact( #VentTimer.Done )
   END_RUNG wire#w15
   RUNG wire#w1
      { S7_Templates := "SrcType := Int" } EQ_Contact(in1 := #StepDelay."Noof StepsPv", in2 := 15)
      wire#w16
      Coil( #ParaOut.Out.LoopValves15 )
   END_RUNG
   RUNG wire#w1
      Contact( #OverTemp )
      Contact( #ParaIn.Selections.VentBeforeOver )
      I_Contact( #VentTimer.Done )
   END_RUNG wire#w16
   RUNG wire#w1
      { S7_Templates := "SrcType := Int" } EQ_Contact(in1 := #StepDelay."Noof StepsPv", in2 := 16)
      wire#w17
      Coil( #ParaOut.Out.LoopValves16 )
   END_RUNG
   RUNG wire#w1
      Contact( #OverTemp )
      Contact( #ParaIn.Selections.VentBeforeOver )
      I_Contact( #VentTimer.Done )
   END_RUNG wire#w17
   RUNG wire#w1
      { S7_Templates := "SrcType := Int" } EQ_Contact(in1 := #StepDelay."Noof StepsPv", in2 := 17)
      wire#w18
      Coil( #ParaOut.Out.LoopValves17 )
   END_RUNG
   RUNG wire#w1
      Contact( #OverTemp )
      Contact( #ParaIn.Selections.VentBeforeOver )
      I_Contact( #VentTimer.Done )
   END_RUNG wire#w18
   // the same network as SCL:
   #_w1 := #CycleRunning AND #CycleEnable AND (#ParaIn.PreciseEngineering.Loops > 0);
   #ParaOut.Out.LoopValves1 := #_w1 AND (((#StepDelay."Noof StepsPv" <= 1) AND NOT #StepDelay.Done AND NOT #VentTimer.Done) OR (#OverTemp AND #ParaIn.Selections.VentBeforeOver AND NOT #VentTimer.Done));
   #ParaOut.Out.LoopValves2 := #_w1 AND ((#StepDelay."Noof StepsPv" = 2) OR (#OverTemp AND #ParaIn.Selections.VentBeforeOver AND NOT #VentTimer.Done));
   #ParaOut.Out.LoopValves3 := #_w1 AND ((#StepDelay."Noof StepsPv" = 3) OR (#OverTemp AND #ParaIn.Selections.VentBeforeOver AND NOT #VentTimer.Done));
   #ParaOut.Out.LoopValves4 := #_w1 AND ((#StepDelay."Noof StepsPv" = 4) OR (#OverTemp AND #ParaIn.Selections.VentBeforeOver AND NOT #VentTimer.Done));
   #ParaOut.Out.LoopValves5 := #_w1 AND ((#StepDelay."Noof StepsPv" = 5) OR (#OverTemp AND #ParaIn.Selections.VentBeforeOver AND NOT #VentTimer.Done));
   #ParaOut.Out.LoopValves6 := #_w1 AND ((#StepDelay."Noof StepsPv" = 6) OR (#OverTemp AND #ParaIn.Selections.VentBeforeOver AND NOT #VentTimer.Done));
   #ParaOut.Out.LoopValves7 := #_w1 AND ((#StepDelay."Noof StepsPv" = 7) OR (#OverTemp AND #ParaIn.Selections.VentBeforeOver AND NOT #VentTimer.Done));
   #ParaOut.Out.LoopValves8 := #_w1 AND ((#StepDelay."Noof StepsPv" = 8) OR (#OverTemp AND #ParaIn.Selections.VentBeforeOver AND NOT #VentTimer.Done));
   #ParaOut.Out.LoopValves9 := #_w1 AND ((#StepDelay."Noof StepsPv" = 9) OR (#OverTemp AND #ParaIn.Selections.VentBeforeOver AND NOT #VentTimer.Done));
   #ParaOut.Out.LoopValves10 := #_w1 AND ((#StepDelay."Noof StepsPv" = 10) OR (#OverTemp AND #ParaIn.Selections.VentBeforeOver AND NOT #VentTimer.Done));
   #ParaOut.Out.LoopValves11 := #_w1 AND ((#StepDelay."Noof StepsPv" = 11) OR (#OverTemp AND #ParaIn.Selections.VentBeforeOver AND NOT #VentTimer.Done));
   #ParaOut.Out.LoopValves12 := #_w1 AND ((#StepDelay."Noof StepsPv" = 12) OR (#OverTemp AND #ParaIn.Selections.VentBeforeOver AND NOT #VentTimer.Done));
   #ParaOut.Out.LoopValves13 := #_w1 AND ((#StepDelay."Noof StepsPv" = 13) OR (#OverTemp AND #ParaIn.Selections.VentBeforeOver AND NOT #VentTimer.Done));
   #ParaOut.Out.LoopValves14 := #_w1 AND ((#StepDelay."Noof StepsPv" = 14) OR (#OverTemp AND #ParaIn.Selections.VentBeforeOver AND NOT #VentTimer.Done));
   #ParaOut.Out.LoopValves15 := #_w1 AND ((#StepDelay."Noof StepsPv" = 15) OR (#OverTemp AND #ParaIn.Selections.VentBeforeOver AND NOT #VentTimer.Done));
   #ParaOut.Out.LoopValves16 := #_w1 AND ((#StepDelay."Noof StepsPv" = 16) OR (#OverTemp AND #ParaIn.Selections.VentBeforeOver AND NOT #VentTimer.Done));
   #ParaOut.Out.LoopValves17 := #_w1 AND ((#StepDelay."Noof StepsPv" = 17) OR (#OverTemp AND #ParaIn.Selections.VentBeforeOver AND NOT #VentTimer.Done));
END_REGION

REGION Network 15: Reset
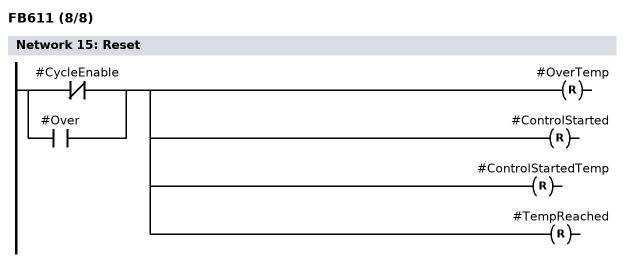
   RUNG wire#powerrail
      I_Contact( #CycleEnable )
      wire#w1
      R_Coil( #OverTemp )
   END_RUNG
   RUNG wire#powerrail
      Contact( #Over )
   END_RUNG wire#w1
   RUNG wire#w1
      R_Coil( #ControlStarted )
   END_RUNG
   RUNG wire#w1
      R_Coil( #ControlStartedTemp )
   END_RUNG
   RUNG wire#w1
      R_Coil( #TempReached )
   END_RUNG
   // the same network as SCL:
   IF NOT #CycleEnable OR #Over THEN
       #OverTemp := FALSE;
       #ControlStarted := FALSE;
       #ControlStartedTemp := FALSE;
       #TempReached := FALSE;
   END_IF;
END_REGION
END_FUNCTION_BLOCK

FUNCTION "FC603" : Void   // FC603, LAD
TITLE = FC603
{ S7_Optimized_Access := 'TRUE' }
// CIP logic
// stored: AutoNumber false, SetENOAutomatically false
   VAR_TEMP
      temp : Int;
      re : Bool;
   END_VAR
   VAR_TEMP   // added for the SCL form of the ladder/FBD networks
      _w1 : Bool;
      _w2 : Bool;
      _w3 : Bool;
   END_VAR
BEGIN

REGION Network 1: NoCycleSelectedInterlock
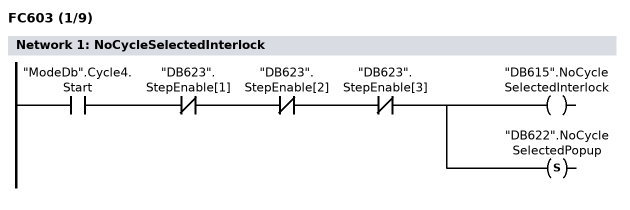
   RUNG wire#powerrail
      Contact( "ModeDb".Cycle4.Start )
      I_Contact( "DB623".StepEnable[1] )
      I_Contact( "DB623".StepEnable[2] )
      I_Contact( "DB623".StepEnable[3] )
      wire#w1
      Coil( "DB615".NoCycleSelectedInterlock )
   END_RUNG
   RUNG wire#w1
      S_Coil( "DB622".NoCycleSelectedPopup )
   END_RUNG
   // the same network as SCL:
   "DB615".NoCycleSelectedInterlock := "ModeDb".Cycle4.Start AND NOT "DB623".StepEnable[1] AND NOT "DB623".StepEnable[2] AND NOT "DB623".StepEnable[3];
   IF "DB615".NoCycleSelectedInterlock THEN "DB622".NoCycleSelectedPopup := TRUE; END_IF;
END_REGION

REGION Network 2: "DB615".Fault
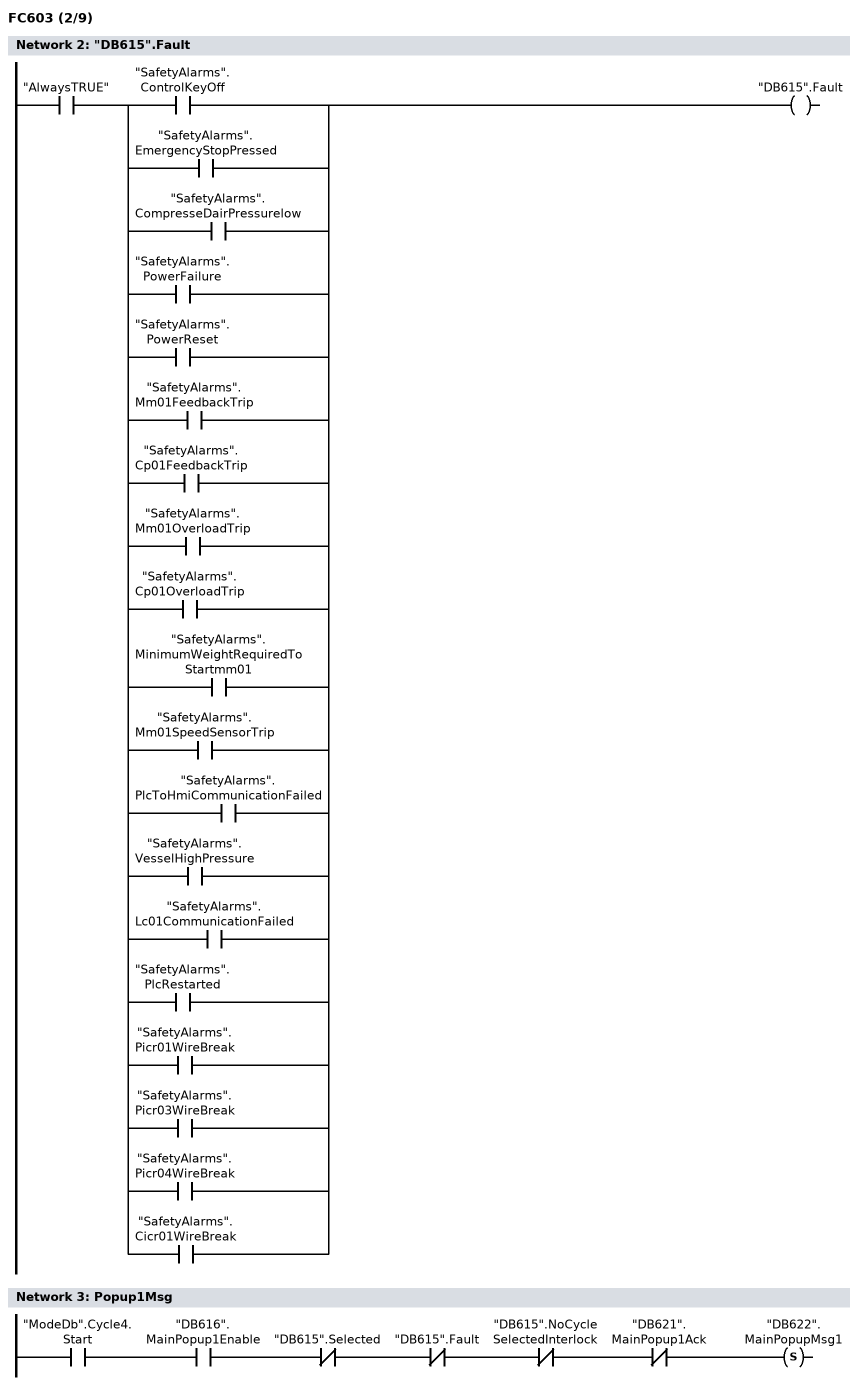
   RUNG wire#powerrail
      Contact( "AlwaysTRUE" )
      wire#w1
      Contact( "SafetyAlarms".ControlKeyOff )
      wire#w2
      Coil( "DB615".Fault )
   END_RUNG
   RUNG wire#w1
      Contact( "SafetyAlarms".EmergencyStopPressed )
   END_RUNG wire#w2
   RUNG wire#w1
      Contact( "SafetyAlarms".CompresseDairPressurelow )
   END_RUNG wire#w2
   RUNG wire#w1
      Contact( "SafetyAlarms".PowerFailure )
   END_RUNG wire#w2
   RUNG wire#w1
      Contact( "SafetyAlarms".PowerReset )
   END_RUNG wire#w2
   RUNG wire#w1
      Contact( "SafetyAlarms".Mm01FeedbackTrip )
   END_RUNG wire#w2
   RUNG wire#w1
      Contact( "SafetyAlarms".Cp01FeedbackTrip )
   END_RUNG wire#w2
   RUNG wire#w1
      Contact( "SafetyAlarms".Mm01OverloadTrip )
   END_RUNG wire#w2
   RUNG wire#w1
      Contact( "SafetyAlarms".Cp01OverloadTrip )
   END_RUNG wire#w2
   RUNG wire#w1
      Contact( "SafetyAlarms".MinimumWeightRequiredToStartmm01 )
   END_RUNG wire#w2
   RUNG wire#w1
      Contact( "SafetyAlarms".Mm01SpeedSensorTrip )
   END_RUNG wire#w2
   RUNG wire#w1
      Contact( "SafetyAlarms".PlcToHmiCommunicationFailed )
   END_RUNG wire#w2
   RUNG wire#w1
      Contact( "SafetyAlarms".VesselHighPressure )
   END_RUNG wire#w2
   RUNG wire#w1
      Contact( "SafetyAlarms".Lc01CommunicationFailed )
   END_RUNG wire#w2
   RUNG wire#w1
      Contact( "SafetyAlarms".PlcRestarted )
   END_RUNG wire#w2
   RUNG wire#w1
      Contact( "SafetyAlarms".Picr01WireBreak )
   END_RUNG wire#w2
   RUNG wire#w1
      Contact( "SafetyAlarms".Picr03WireBreak )
   END_RUNG wire#w2
   RUNG wire#w1
      Contact( "SafetyAlarms".Picr04WireBreak )
   END_RUNG wire#w2
   RUNG wire#w1
      Contact( "SafetyAlarms".Cicr01WireBreak )
   END_RUNG wire#w2
   // the same network as SCL:
   "DB615".Fault := "AlwaysTRUE" AND ("SafetyAlarms".ControlKeyOff OR "SafetyAlarms".EmergencyStopPressed OR "SafetyAlarms".CompresseDairPressurelow OR "SafetyAlarms".PowerFailure OR "SafetyAlarms".PowerReset OR "SafetyAlarms".Mm01FeedbackTrip OR "SafetyAlarms".Cp01FeedbackTrip OR "SafetyAlarms".Mm01OverloadTrip OR "SafetyAlarms".Cp01OverloadTrip OR "SafetyAlarms".MinimumWeightRequiredToStartmm01 OR "SafetyAlarms".Mm01SpeedSensorTrip OR "SafetyAlarms".PlcToHmiCommunicationFailed OR "SafetyAlarms".VesselHighPressure OR "SafetyAlarms".Lc01CommunicationFailed OR "SafetyAlarms".PlcRestarted OR "SafetyAlarms".Picr01WireBreak OR "SafetyAlarms".Picr03WireBreak OR "SafetyAlarms".Picr04WireBreak OR "SafetyAlarms".Cicr01WireBreak);
END_REGION

REGION Network 3: Popup1Msg
   RUNG wire#powerrail
      Contact( "ModeDb".Cycle4.Start )
      Contact( "DB616".MainPopup1Enable )
      I_Contact( "DB615".Selected )
      I_Contact( "DB615".Fault )
      I_Contact( "DB615".NoCycleSelectedInterlock )
      I_Contact( "DB621".MainPopup1Ack )
      S_Coil( "DB622".MainPopupMsg1 )
   END_RUNG
   // the same network as SCL:
   IF "ModeDb".Cycle4.Start AND "DB616".MainPopup1Enable AND NOT "DB615".Selected AND NOT "DB615".Fault AND NOT "DB615".NoCycleSelectedInterlock AND NOT "DB621".MainPopup1Ack THEN
       "DB622".MainPopupMsg1 := TRUE;
   END_IF;
END_REGION

REGION Network 4: Popup2Msg
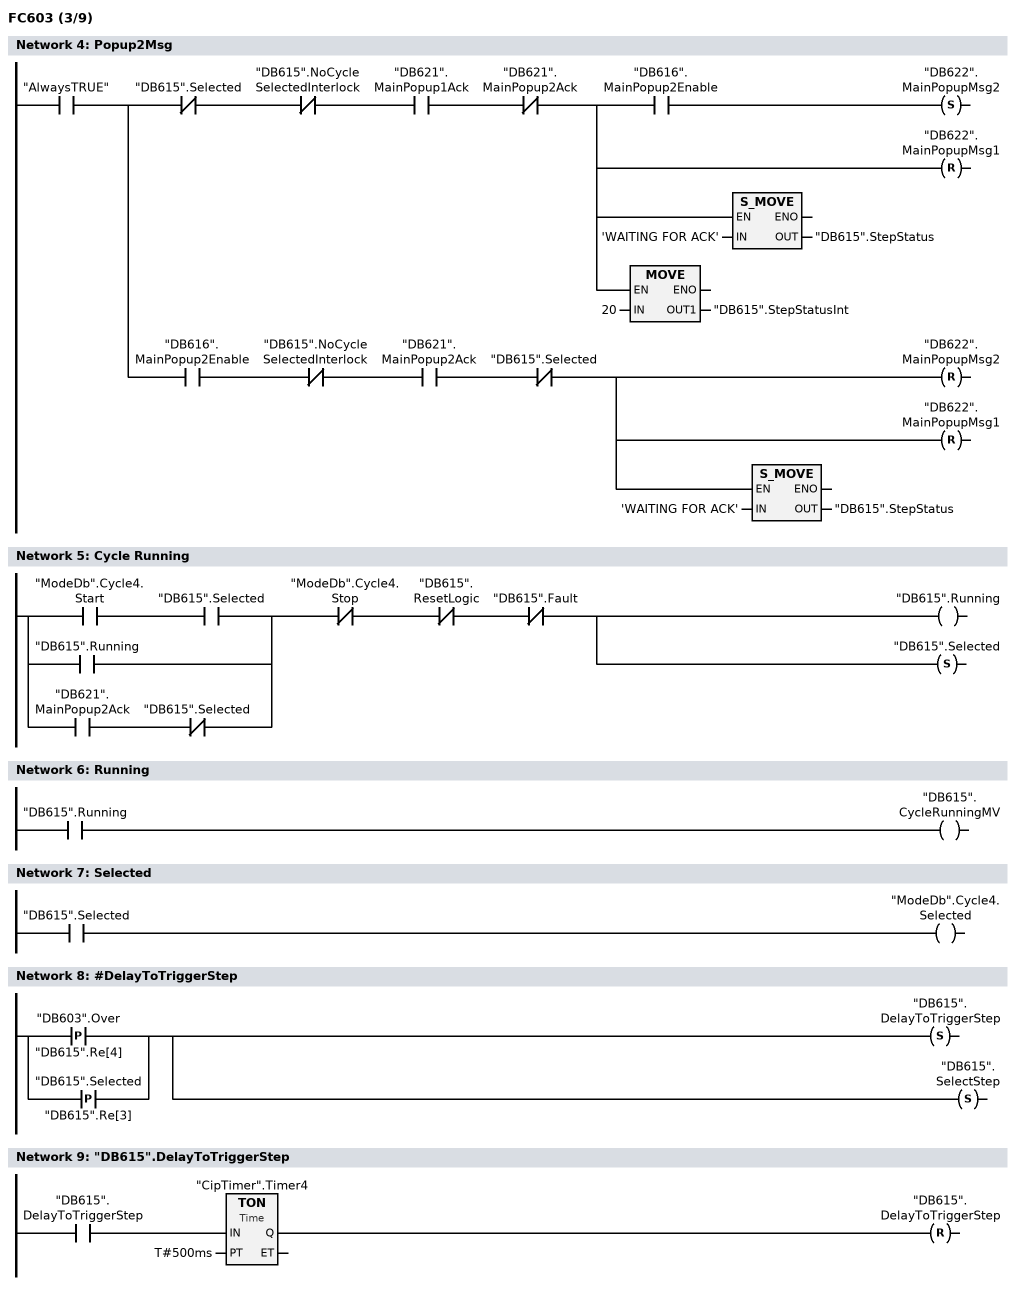
   RUNG wire#powerrail
      Contact( "AlwaysTRUE" )
      wire#w1
      I_Contact( "DB615".Selected )
      I_Contact( "DB615".NoCycleSelectedInterlock )
      Contact( "DB621".MainPopup1Ack )
      I_Contact( "DB621".MainPopup2Ack )
      wire#w2
      Contact( "DB616".MainPopup2Enable )
      S_Coil( "DB622".MainPopupMsg2 )
   END_RUNG
   RUNG wire#w2
      R_Coil( "DB622".MainPopupMsg1 )
   END_RUNG
   RUNG wire#w2
      S_Move(in := 'WAITING FOR ACK', out => "DB615".StepStatus)
   END_RUNG
   RUNG wire#w2
      Move(in := 20, out1 => "DB615".StepStatusInt)
   END_RUNG
   RUNG wire#w1
      Contact( "DB616".MainPopup2Enable )
      I_Contact( "DB615".NoCycleSelectedInterlock )
      Contact( "DB621".MainPopup2Ack )
      I_Contact( "DB615".Selected )
      wire#w3
      R_Coil( "DB622".MainPopupMsg2 )
   END_RUNG
   RUNG wire#w3
      R_Coil( "DB622".MainPopupMsg1 )
   END_RUNG
   RUNG wire#w3
      S_Move(in := 'WAITING FOR ACK', out => "DB615".StepStatus)
   END_RUNG
   // the same network as SCL:
   #_w1 := "AlwaysTRUE" AND NOT "DB615".Selected AND NOT "DB615".NoCycleSelectedInterlock AND "DB621".MainPopup1Ack AND NOT "DB621".MainPopup2Ack;
   IF #_w1 AND "DB616".MainPopup2Enable THEN "DB622".MainPopupMsg2 := TRUE; END_IF;
   IF #_w1 THEN
       "DB622".MainPopupMsg1 := FALSE;
       "DB615".StepStatus := 'WAITING FOR ACK';
       "DB615".StepStatusInt := 20;
   END_IF;
   IF "AlwaysTRUE" AND "DB616".MainPopup2Enable AND NOT "DB615".NoCycleSelectedInterlock AND "DB621".MainPopup2Ack AND NOT "DB615".Selected THEN
       "DB622".MainPopupMsg2 := FALSE;
       "DB622".MainPopupMsg1 := FALSE;
       "DB615".StepStatus := 'WAITING FOR ACK';
   END_IF;
END_REGION

REGION Network 5: Cycle Running
   RUNG wire#powerrail
      Contact( "ModeDb".Cycle4.Start )
      Contact( "DB615".Selected )
      wire#w1
      I_Contact( "ModeDb".Cycle4.Stop )
      I_Contact( "DB615".ResetLogic )
      I_Contact( "DB615".Fault )
      wire#w2
      Coil( "DB615".Running )
   END_RUNG
   RUNG wire#powerrail
      Contact( "DB615".Running )
   END_RUNG wire#w1
   RUNG wire#powerrail
      Contact( "DB621".MainPopup2Ack )
      I_Contact( "DB615".Selected )
   END_RUNG wire#w1
   RUNG wire#w2
      S_Coil( "DB615".Selected )
   END_RUNG
   // the same network as SCL:
   "DB615".Running := (("ModeDb".Cycle4.Start AND "DB615".Selected) OR "DB615".Running OR ("DB621".MainPopup2Ack AND NOT "DB615".Selected)) AND NOT "ModeDb".Cycle4.Stop AND NOT "DB615".ResetLogic AND NOT "DB615".Fault;
   IF "DB615".Running THEN "DB615".Selected := TRUE; END_IF;
END_REGION

REGION Network 6: Running
   RUNG wire#powerrail
      Contact( "DB615".Running )
      Coil( "DB615".CycleRunningMV )
   END_RUNG
   // the same network as SCL:
   "DB615".CycleRunningMV := "DB615".Running;
END_REGION

REGION Network 7: Selected
   RUNG wire#powerrail
      Contact( "DB615".Selected )
      Coil( "ModeDb".Cycle4.Selected )
   END_RUNG
   // the same network as SCL:
   "ModeDb".Cycle4.Selected := "DB615".Selected;
END_REGION

REGION Network 8: #DelayToTriggerStep
   RUNG wire#powerrail
      P_Contact(operand := "DB603".Over, bit := "DB615".Re[4])
      wire#w1
      S_Coil( "DB615".DelayToTriggerStep )
   END_RUNG
   RUNG wire#powerrail
      P_Contact(operand := "DB615".Selected, bit := "DB615".Re[3])
   END_RUNG wire#w1
   RUNG wire#w1
      S_Coil( "DB615".SelectStep )
   END_RUNG
   // the same network as SCL:
   #_w1 := "DB603".Over AND NOT "DB615".Re[4];   // rising edge of "DB603".Over
   "DB615".Re[4] := "DB603".Over;
   #_w2 := "DB615".Selected AND NOT "DB615".Re[3];   // rising edge of "DB615".Selected
   "DB615".Re[3] := "DB615".Selected;
   IF #_w1 OR #_w2 THEN
       "DB615".DelayToTriggerStep := TRUE;
       "DB615".SelectStep := TRUE;
   END_IF;
END_REGION

REGION Network 9: "DB615".DelayToTriggerStep
   RUNG wire#powerrail
      Contact( "DB615".DelayToTriggerStep )
      { S7_Templates := "time_type := Time" } "CipTimer".Timer4.TON(pt := T#500ms, et =>)
      R_Coil( "DB615".DelayToTriggerStep )
   END_RUNG
   // the same network as SCL:
   "CipTimer".Timer4.TON(IN := "DB615".DelayToTriggerStep, PT := T#500ms);
   IF "CipTimer".Timer4.Q THEN "DB615".DelayToTriggerStep := FALSE; END_IF;
END_REGION

REGION Network 10: CYCLE STATUS
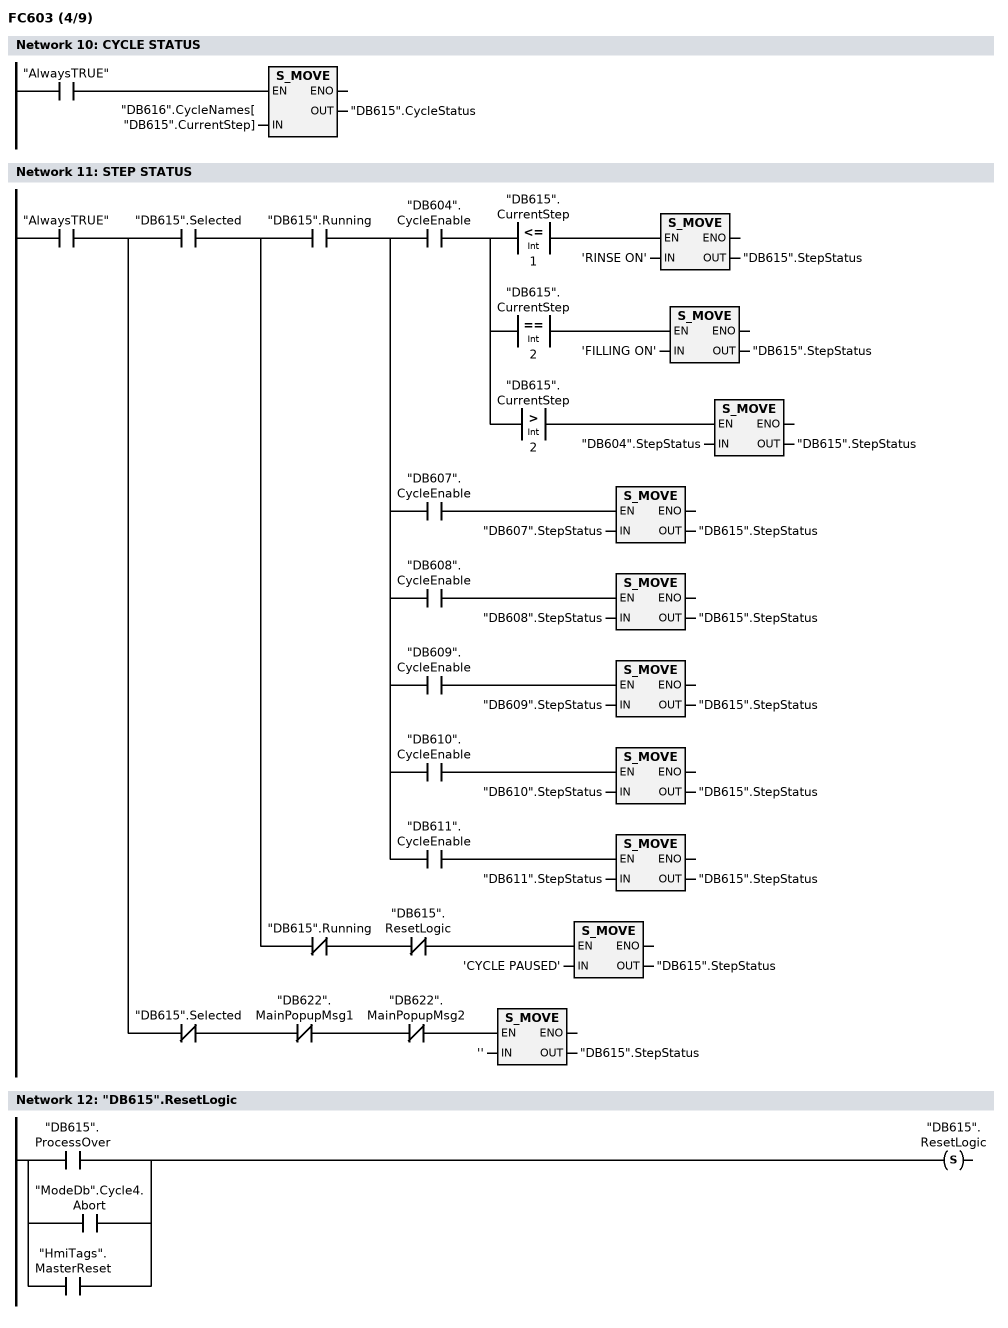
   RUNG wire#powerrail
      Contact( "AlwaysTRUE" )
      S_Move(in := "DB616".CycleNames["DB615".CurrentStep], out => "DB615".CycleStatus)
   END_RUNG
   // the same network as SCL:
   IF "AlwaysTRUE" THEN "DB615".CycleStatus := "DB616".CycleNames["DB615".CurrentStep]; END_IF;
END_REGION

REGION Network 11: STEP STATUS
   RUNG wire#powerrail
      Contact( "AlwaysTRUE" )
      wire#w1
      Contact( "DB615".Selected )
      wire#w2
      Contact( "DB615".Running )
      wire#w3
      Contact( "DB604".CycleEnable )
      wire#w4
      { S7_Templates := "SrcType := Int" } LE_Contact(in1 := "DB615".CurrentStep, in2 := 1)
      S_Move(in := 'RINSE ON', out => "DB615".StepStatus)
   END_RUNG
   RUNG wire#w4
      { S7_Templates := "SrcType := Int" } EQ_Contact(in1 := "DB615".CurrentStep, in2 := 2)
      S_Move(in := 'FILLING ON', out => "DB615".StepStatus)
   END_RUNG
   RUNG wire#w4
      { S7_Templates := "SrcType := Int" } GT_Contact(in1 := "DB615".CurrentStep, in2 := 2)
      S_Move(in := "DB604".StepStatus, out => "DB615".StepStatus)
   END_RUNG
   RUNG wire#w3
      Contact( "DB607".CycleEnable )
      S_Move(in := "DB607".StepStatus, out => "DB615".StepStatus)
   END_RUNG
   RUNG wire#w3
      Contact( "DB608".CycleEnable )
      S_Move(in := "DB608".StepStatus, out => "DB615".StepStatus)
   END_RUNG
   RUNG wire#w3
      Contact( "DB609".CycleEnable )
      S_Move(in := "DB609".StepStatus, out => "DB615".StepStatus)
   END_RUNG
   RUNG wire#w3
      Contact( "DB610".CycleEnable )
      S_Move(in := "DB610".StepStatus, out => "DB615".StepStatus)
   END_RUNG
   RUNG wire#w3
      Contact( "DB611".CycleEnable )
      S_Move(in := "DB611".StepStatus, out => "DB615".StepStatus)
   END_RUNG
   RUNG wire#w2
      I_Contact( "DB615".Running )
      I_Contact( "DB615".ResetLogic )
      S_Move(in := 'CYCLE PAUSED', out => "DB615".StepStatus)
   END_RUNG
   RUNG wire#w1
      I_Contact( "DB615".Selected )
      I_Contact( "DB622".MainPopupMsg1 )
      I_Contact( "DB622".MainPopupMsg2 )
      S_Move(in := '', out => "DB615".StepStatus)
   END_RUNG
   // the same network as SCL:
   #_w1 := "AlwaysTRUE" AND "DB615".Selected;
   #_w2 := #_w1 AND "DB615".Running;
   #_w3 := #_w2 AND "DB604".CycleEnable;
   IF #_w3 AND ("DB615".CurrentStep <= 1) THEN "DB615".StepStatus := 'RINSE ON'; END_IF;
   IF #_w3 AND ("DB615".CurrentStep = 2) THEN "DB615".StepStatus := 'FILLING ON'; END_IF;
   IF #_w3 AND ("DB615".CurrentStep > 2) THEN "DB615".StepStatus := "DB604".StepStatus; END_IF;
   IF #_w2 AND "DB607".CycleEnable THEN "DB615".StepStatus := "DB607".StepStatus; END_IF;
   IF #_w2 AND "DB608".CycleEnable THEN "DB615".StepStatus := "DB608".StepStatus; END_IF;
   IF #_w2 AND "DB609".CycleEnable THEN "DB615".StepStatus := "DB609".StepStatus; END_IF;
   IF #_w2 AND "DB610".CycleEnable THEN "DB615".StepStatus := "DB610".StepStatus; END_IF;
   IF #_w2 AND "DB611".CycleEnable THEN "DB615".StepStatus := "DB611".StepStatus; END_IF;
   IF #_w1 AND NOT "DB615".Running AND NOT "DB615".ResetLogic THEN
       "DB615".StepStatus := 'CYCLE PAUSED';
   END_IF;
   IF "AlwaysTRUE" AND NOT "DB615".Selected AND NOT "DB622".MainPopupMsg1 AND NOT "DB622".MainPopupMsg2 THEN
       "DB615".StepStatus := '';
   END_IF;
END_REGION

REGION Network 12: "DB615".ResetLogic
   RUNG wire#powerrail
      Contact( "DB615".ProcessOver )
      wire#w1
      S_Coil( "DB615".ResetLogic )
   END_RUNG
   RUNG wire#powerrail
      Contact( "ModeDb".Cycle4.Abort )
   END_RUNG wire#w1
   RUNG wire#powerrail
      Contact( "HmiTags".MasterReset )
   END_RUNG wire#w1
   // the same network as SCL:
   IF "DB615".ProcessOver OR "ModeDb".Cycle4.Abort OR "HmiTags".MasterReset THEN
       "DB615".ResetLogic := TRUE;
   END_IF;
END_REGION

REGION Network 13: "Printing".ResultCip
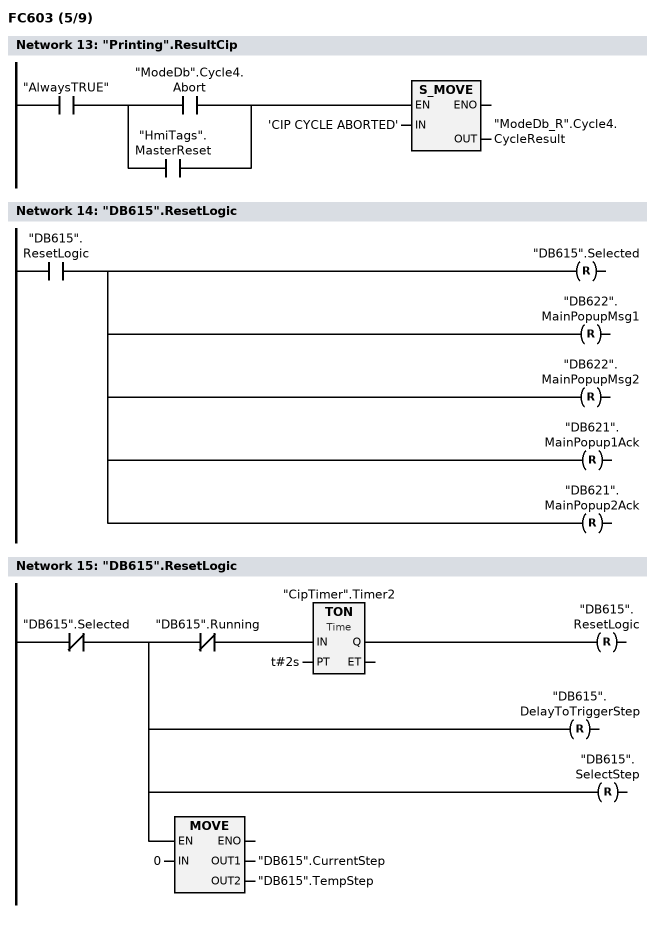
   RUNG wire#powerrail
      Contact( "AlwaysTRUE" )
      wire#w1
      Contact( "ModeDb".Cycle4.Abort )
      wire#w2
      S_Move(in := 'CIP CYCLE ABORTED', out => "ModeDb_R".Cycle4.CycleResult)
   END_RUNG
   RUNG wire#w1
      Contact( "HmiTags".MasterReset )
   END_RUNG wire#w2
   // the same network as SCL:
   IF "AlwaysTRUE" AND ("ModeDb".Cycle4.Abort OR "HmiTags".MasterReset) THEN
       "ModeDb_R".Cycle4.CycleResult := 'CIP CYCLE ABORTED';
   END_IF;
END_REGION

REGION Network 14: "DB615".ResetLogic
   RUNG wire#powerrail
      Contact( "DB615".ResetLogic )
      wire#w1
      R_Coil( "DB615".Selected )
   END_RUNG
   RUNG wire#w1
      R_Coil( "DB622".MainPopupMsg1 )
   END_RUNG
   RUNG wire#w1
      R_Coil( "DB622".MainPopupMsg2 )
   END_RUNG
   RUNG wire#w1
      R_Coil( "DB621".MainPopup1Ack )
   END_RUNG
   RUNG wire#w1
      R_Coil( "DB621".MainPopup2Ack )
   END_RUNG
   // the same network as SCL:
   IF "DB615".ResetLogic THEN
       "DB615".Selected := FALSE;
       "DB622".MainPopupMsg1 := FALSE;
       "DB622".MainPopupMsg2 := FALSE;
       "DB621".MainPopup1Ack := FALSE;
       "DB621".MainPopup2Ack := FALSE;
   END_IF;
END_REGION

REGION Network 15: "DB615".ResetLogic
   RUNG wire#powerrail
      I_Contact( "DB615".Selected )
      wire#w1
      I_Contact( "DB615".Running )
      { S7_Templates := "time_type := Time" } "CipTimer".Timer2.TON(pt := t#2s, et =>)
      R_Coil( "DB615".ResetLogic )
   END_RUNG
   RUNG wire#w1
      R_Coil( "DB615".DelayToTriggerStep )
   END_RUNG
   RUNG wire#w1
      R_Coil( "DB615".SelectStep )
   END_RUNG
   RUNG wire#w1
      Move(in := 0, out1 => "DB615".CurrentStep, out2 => "DB615".TempStep)
   END_RUNG
   // the same network as SCL:
   "CipTimer".Timer2.TON(IN := NOT "DB615".Selected AND NOT "DB615".Running, PT := t#2s);
   IF "CipTimer".Timer2.Q THEN "DB615".ResetLogic := FALSE; END_IF;
   IF NOT "DB615".Selected THEN
       "DB615".DelayToTriggerStep := FALSE;
       "DB615".SelectStep := FALSE;
       "DB615".CurrentStep := 0;
       "DB615".TempStep := 0;
   END_IF;
END_REGION

REGION Network 16: Button Reset
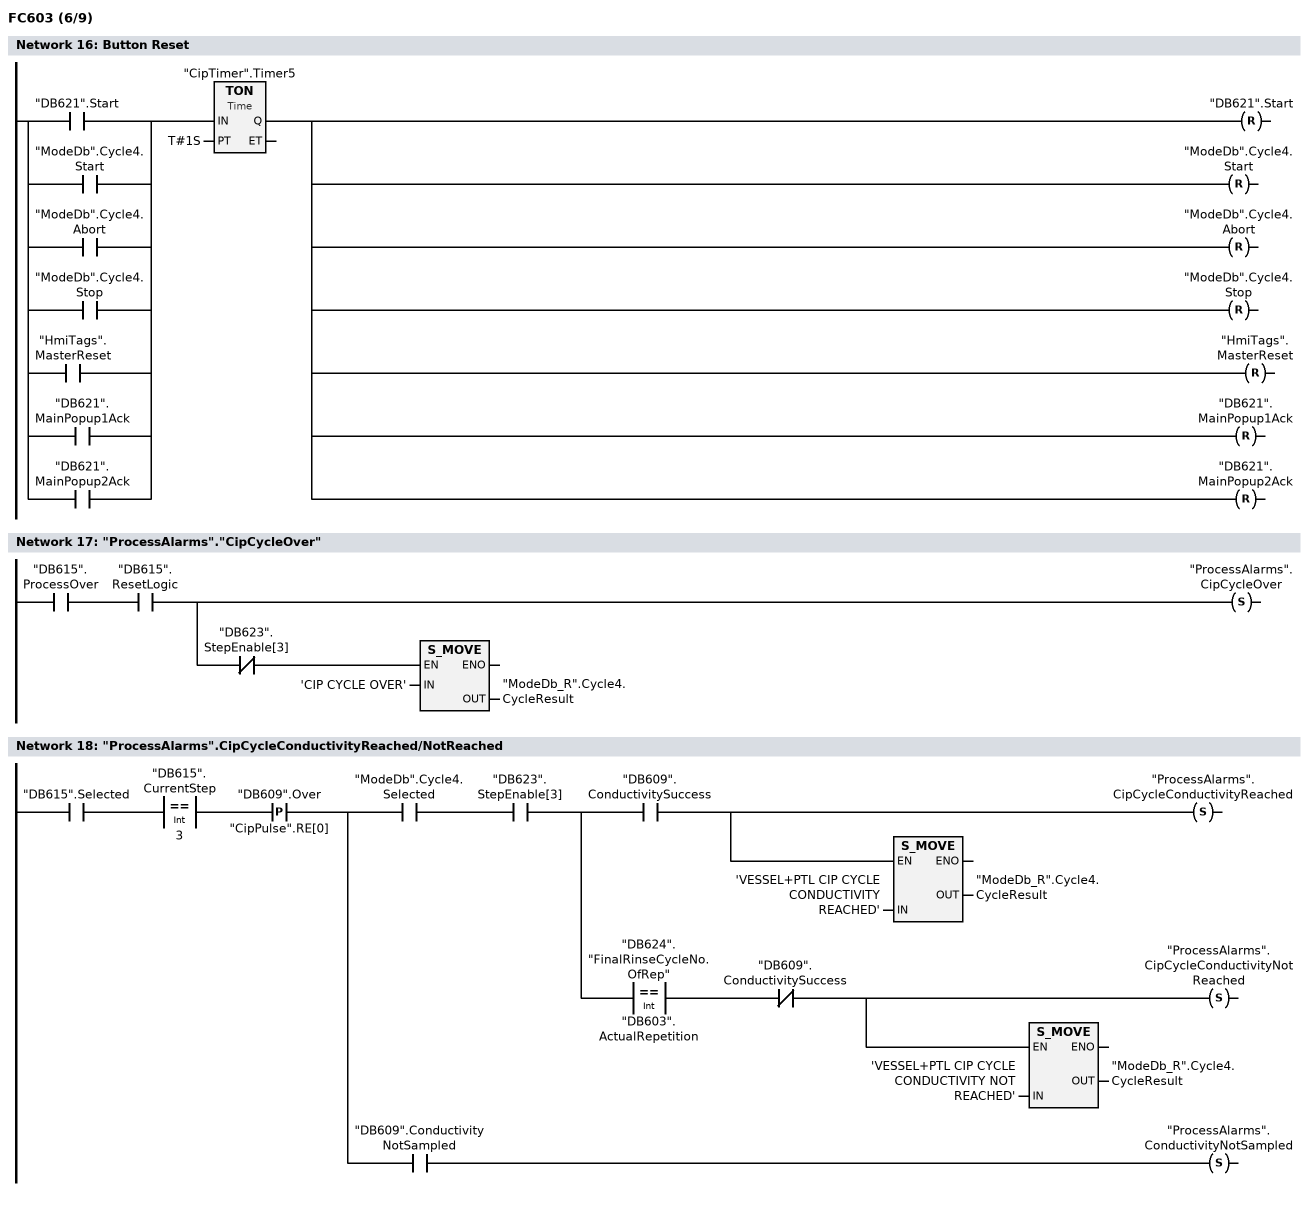
   RUNG wire#powerrail
      Contact( "DB621".Start )
      wire#w1
      { S7_Templates := "time_type := Time" } "CipTimer".Timer5.TON(pt := T#1S, et =>)
      wire#w2
      R_Coil( "DB621".Start )
   END_RUNG
   RUNG wire#powerrail
      Contact( "ModeDb".Cycle4.Start )
   END_RUNG wire#w1
   RUNG wire#powerrail
      Contact( "ModeDb".Cycle4.Abort )
   END_RUNG wire#w1
   RUNG wire#powerrail
      Contact( "ModeDb".Cycle4.Stop )
   END_RUNG wire#w1
   RUNG wire#powerrail
      Contact( "HmiTags".MasterReset )
   END_RUNG wire#w1
   RUNG wire#powerrail
      Contact( "DB621".MainPopup1Ack )
   END_RUNG wire#w1
   RUNG wire#powerrail
      Contact( "DB621".MainPopup2Ack )
   END_RUNG wire#w1
   RUNG wire#w2
      R_Coil( "ModeDb".Cycle4.Start )
   END_RUNG
   RUNG wire#w2
      R_Coil( "ModeDb".Cycle4.Abort )
   END_RUNG
   RUNG wire#w2
      R_Coil( "ModeDb".Cycle4.Stop )
   END_RUNG
   RUNG wire#w2
      R_Coil( "HmiTags".MasterReset )
   END_RUNG
   RUNG wire#w2
      R_Coil( "DB621".MainPopup1Ack )
   END_RUNG
   RUNG wire#w2
      R_Coil( "DB621".MainPopup2Ack )
   END_RUNG
   // the same network as SCL:
   "CipTimer".Timer5.TON(IN := "DB621".Start OR "ModeDb".Cycle4.Start OR "ModeDb".Cycle4.Abort OR "ModeDb".Cycle4.Stop OR "HmiTags".MasterReset OR "DB621".MainPopup1Ack OR "DB621".MainPopup2Ack,
                         PT := T#1S);
   IF "CipTimer".Timer5.Q THEN
       "DB621".Start := FALSE;
       "ModeDb".Cycle4.Start := FALSE;
       "ModeDb".Cycle4.Abort := FALSE;
       "ModeDb".Cycle4.Stop := FALSE;
       "HmiTags".MasterReset := FALSE;
       "DB621".MainPopup1Ack := FALSE;
       "DB621".MainPopup2Ack := FALSE;
   END_IF;
END_REGION

REGION Network 17: "ProcessAlarms"."CipCycleOver"
   RUNG wire#powerrail
      Contact( "DB615".ProcessOver )
      Contact( "DB615".ResetLogic )
      wire#w1
      S_Coil( "ProcessAlarms".CipCycleOver )
   END_RUNG
   RUNG wire#w1
      I_Contact( "DB623".StepEnable[3] )
      S_Move(in := 'CIP CYCLE OVER', out => "ModeDb_R".Cycle4.CycleResult)
   END_RUNG
   // the same network as SCL:
   #_w1 := "DB615".ProcessOver AND "DB615".ResetLogic;
   IF #_w1 THEN "ProcessAlarms".CipCycleOver := TRUE; END_IF;
   IF #_w1 AND NOT "DB623".StepEnable[3] THEN "ModeDb_R".Cycle4.CycleResult := 'CIP CYCLE OVER'; END_IF;
END_REGION

REGION Network 18: "ProcessAlarms".CipCycleConductivityReached/NotReached
   RUNG wire#powerrail
      Contact( "DB615".Selected )
      { S7_Templates := "SrcType := Int" } EQ_Contact(in1 := "DB615".CurrentStep, in2 := 3)
      P_Contact(operand := "DB609".Over, bit := "CipPulse".RE[0])
      wire#w1
      Contact( "ModeDb".Cycle4.Selected )
      Contact( "DB623".StepEnable[3] )
      wire#w2
      Contact( "DB609".ConductivitySuccess )
      wire#w3
      S_Coil( "ProcessAlarms".CipCycleConductivityReached )
   END_RUNG
   RUNG wire#w3
      S_Move(in := 'VESSEL+PTL CIP CYCLE CONDUCTIVITY REACHED', out => "ModeDb_R".Cycle4.CycleResult)
   END_RUNG
   RUNG wire#w2
      { S7_Templates := "SrcType := Int" } EQ_Contact(in1 := "DB624"."FinalRinseCycleNo.OfRep", in2 := "DB603".ActualRepetition)
      I_Contact( "DB609".ConductivitySuccess )
      wire#w4
      S_Coil( "ProcessAlarms".CipCycleConductivityNotReached )
   END_RUNG
   RUNG wire#w4
      S_Move(in := 'VESSEL+PTL CIP CYCLE CONDUCTIVITY NOT REACHED', out => "ModeDb_R".Cycle4.CycleResult)
   END_RUNG
   RUNG wire#w1
      Contact( "DB609".ConductivityNotSampled )
      S_Coil( "ProcessAlarms".ConductivityNotSampled )
   END_RUNG
   // the same network as SCL:
   #_w1 := "DB615".Selected AND ("DB615".CurrentStep = 3) AND "DB609".Over AND NOT "CipPulse".RE[0];   // rising edge of "DB609".Over
   "CipPulse".RE[0] := "DB609".Over;
   #_w2 := #_w1 AND "ModeDb".Cycle4.Selected AND "DB623".StepEnable[3];
   IF #_w2 AND "DB609".ConductivitySuccess THEN
       "ProcessAlarms".CipCycleConductivityReached := TRUE;
       "ModeDb_R".Cycle4.CycleResult := 'VESSEL+PTL CIP CYCLE CONDUCTIVITY REACHED';
   END_IF;
   IF #_w2 AND ("DB624"."FinalRinseCycleNo.OfRep" = "DB603".ActualRepetition) AND NOT "DB609".ConductivitySuccess THEN
       "ProcessAlarms".CipCycleConductivityNotReached := TRUE;
       "ModeDb_R".Cycle4.CycleResult := 'VESSEL+PTL CIP CYCLE CONDUCTIVITY NOT REACHED';
   END_IF;
   IF #_w1 AND "DB609".ConductivityNotSampled THEN "ProcessAlarms".ConductivityNotSampled := TRUE; END_IF;
END_REGION

REGION Network 19: "HmiTags".AlarmAck
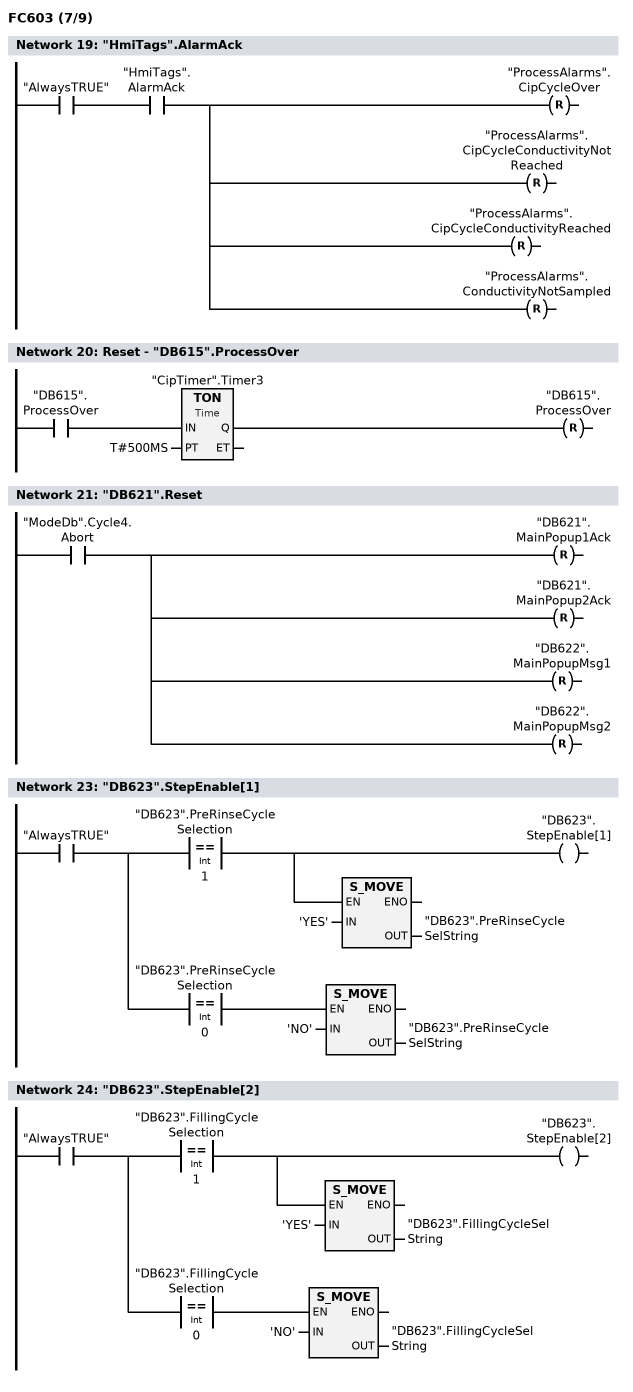
   RUNG wire#powerrail
      Contact( "AlwaysTRUE" )
      Contact( "HmiTags".AlarmAck )
      wire#w1
      R_Coil( "ProcessAlarms".CipCycleOver )
   END_RUNG
   RUNG wire#w1
      R_Coil( "ProcessAlarms".CipCycleConductivityNotReached )
   END_RUNG
   RUNG wire#w1
      R_Coil( "ProcessAlarms".CipCycleConductivityReached )
   END_RUNG
   RUNG wire#w1
      R_Coil( "ProcessAlarms".ConductivityNotSampled )
   END_RUNG
   // the same network as SCL:
   IF "AlwaysTRUE" AND "HmiTags".AlarmAck THEN
       "ProcessAlarms".CipCycleOver := FALSE;
       "ProcessAlarms".CipCycleConductivityNotReached := FALSE;
       "ProcessAlarms".CipCycleConductivityReached := FALSE;
       "ProcessAlarms".ConductivityNotSampled := FALSE;
   END_IF;
END_REGION

REGION Network 20: Reset - "DB615".ProcessOver
   RUNG wire#powerrail
      Contact( "DB615".ProcessOver )
      { S7_Templates := "time_type := Time" } "CipTimer".Timer3.TON(pt := T#500MS, et =>)
      R_Coil( "DB615".ProcessOver )
   END_RUNG
   // the same network as SCL:
   "CipTimer".Timer3.TON(IN := "DB615".ProcessOver, PT := T#500MS);
   IF "CipTimer".Timer3.Q THEN "DB615".ProcessOver := FALSE; END_IF;
END_REGION

REGION Network 21: "DB621".Reset
   RUNG wire#powerrail
      Contact( "ModeDb".Cycle4.Abort )
      wire#w1
      R_Coil( "DB621".MainPopup1Ack )
   END_RUNG
   RUNG wire#w1
      R_Coil( "DB621".MainPopup2Ack )
   END_RUNG
   RUNG wire#w1
      R_Coil( "DB622".MainPopupMsg1 )
   END_RUNG
   RUNG wire#w1
      R_Coil( "DB622".MainPopupMsg2 )
   END_RUNG
   // the same network as SCL:
   IF "ModeDb".Cycle4.Abort THEN
       "DB621".MainPopup1Ack := FALSE;
       "DB621".MainPopup2Ack := FALSE;
       "DB622".MainPopupMsg1 := FALSE;
       "DB622".MainPopupMsg2 := FALSE;
   END_IF;
END_REGION

REGION Network 22: *********MV 3000 *****************
END_REGION

REGION Network 23: "DB623".StepEnable[1]
   RUNG wire#powerrail
      Contact( "AlwaysTRUE" )
      wire#w1
      { S7_Templates := "SrcType := Int" } EQ_Contact(in1 := "DB623".PreRinseCycleSelection, in2 := 1)
      wire#w2
      Coil( "DB623".StepEnable[1] )
   END_RUNG
   RUNG wire#w2
      S_Move(in := 'YES', out => "DB623".PreRinseCycleSelString)
   END_RUNG
   RUNG wire#w1
      { S7_Templates := "SrcType := Int" } EQ_Contact(in1 := "DB623".PreRinseCycleSelection, in2 := 0)
      S_Move(in := 'NO', out => "DB623".PreRinseCycleSelString)
   END_RUNG
   // the same network as SCL:
   "DB623".StepEnable[1] := "AlwaysTRUE" AND ("DB623".PreRinseCycleSelection = 1);
   IF "AlwaysTRUE" AND ("DB623".PreRinseCycleSelection = 1) THEN
       "DB623".PreRinseCycleSelString := 'YES';
   END_IF;
   IF "AlwaysTRUE" AND ("DB623".PreRinseCycleSelection = 0) THEN
       "DB623".PreRinseCycleSelString := 'NO';
   END_IF;
END_REGION

REGION Network 24: "DB623".StepEnable[2]
   RUNG wire#powerrail
      Contact( "AlwaysTRUE" )
      wire#w1
      { S7_Templates := "SrcType := Int" } EQ_Contact(in1 := "DB623".FillingCycleSelection, in2 := 1)
      wire#w2
      Coil( "DB623".StepEnable[2] )
   END_RUNG
   RUNG wire#w2
      S_Move(in := 'YES', out => "DB623".FillingCycleSelString)
   END_RUNG
   RUNG wire#w1
      { S7_Templates := "SrcType := Int" } EQ_Contact(in1 := "DB623".FillingCycleSelection, in2 := 0)
      S_Move(in := 'NO', out => "DB623".FillingCycleSelString)
   END_RUNG
   // the same network as SCL:
   "DB623".StepEnable[2] := "AlwaysTRUE" AND ("DB623".FillingCycleSelection = 1);
   IF "AlwaysTRUE" AND ("DB623".FillingCycleSelection = 1) THEN
       "DB623".FillingCycleSelString := 'YES';
   END_IF;
   IF "AlwaysTRUE" AND ("DB623".FillingCycleSelection = 0) THEN
       "DB623".FillingCycleSelString := 'NO';
   END_IF;
END_REGION

REGION Network 25: "DB623".StepEnable[3]
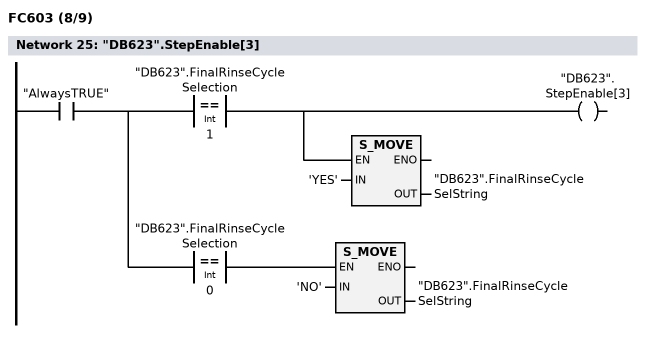
   RUNG wire#powerrail
      Contact( "AlwaysTRUE" )
      wire#w1
      { S7_Templates := "SrcType := Int" } EQ_Contact(in1 := "DB623".FinalRinseCycleSelection, in2 := 1)
      wire#w2
      Coil( "DB623".StepEnable[3] )
   END_RUNG
   RUNG wire#w2
      S_Move(in := 'YES', out => "DB623".FinalRinseCycleSelString)
   END_RUNG
   RUNG wire#w1
      { S7_Templates := "SrcType := Int" } EQ_Contact(in1 := "DB623".FinalRinseCycleSelection, in2 := 0)
      S_Move(in := 'NO', out => "DB623".FinalRinseCycleSelString)
   END_RUNG
   // the same network as SCL:
   "DB623".StepEnable[3] := "AlwaysTRUE" AND ("DB623".FinalRinseCycleSelection = 1);
   IF "AlwaysTRUE" AND ("DB623".FinalRinseCycleSelection = 1) THEN
       "DB623".FinalRinseCycleSelString := 'YES';
   END_IF;
   IF "AlwaysTRUE" AND ("DB623".FinalRinseCycleSelection = 0) THEN
       "DB623".FinalRinseCycleSelString := 'NO';
   END_IF;
END_REGION

REGION Network 27: Para Passing of AP AI sensor
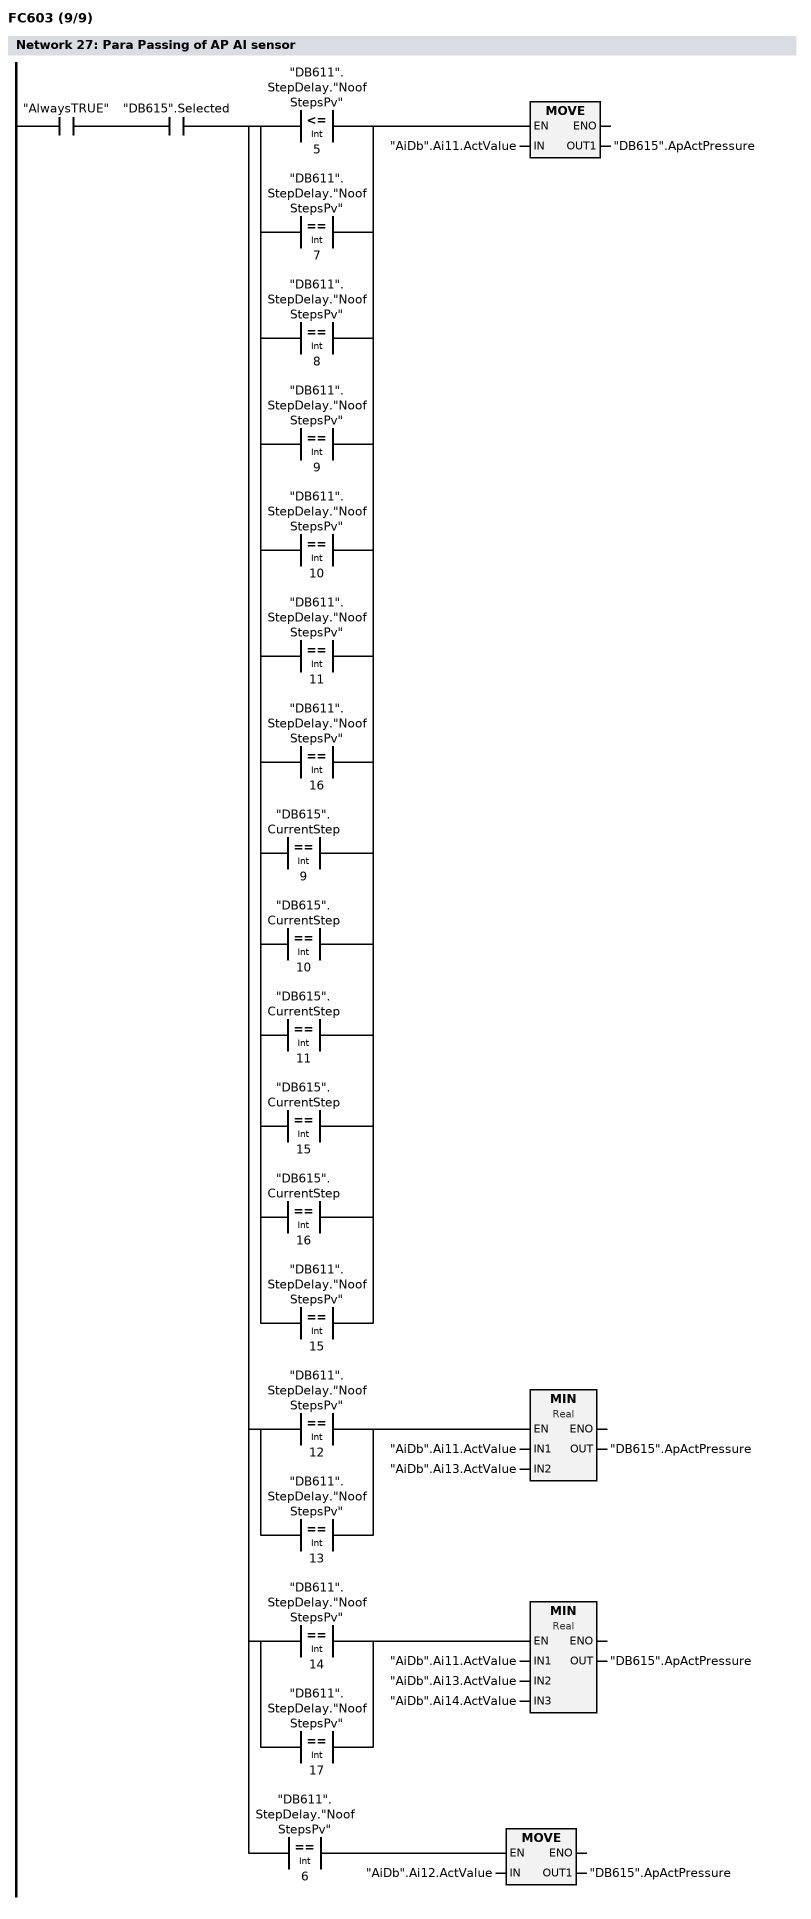
   RUNG wire#powerrail
      Contact( "AlwaysTRUE" )
      Contact( "DB615".Selected )
      wire#w1
      { S7_Templates := "SrcType := Int" } LE_Contact(in1 := "DB611".StepDelay."Noof StepsPv", in2 := 5)
      wire#w2
      Move(in := "AiDb".Ai11.ActValue, out1 => "DB615".ApActPressure)
   END_RUNG
   RUNG wire#w1
      { S7_Templates := "SrcType := Int" } EQ_Contact(in1 := "DB611".StepDelay."Noof StepsPv", in2 := 7)
   END_RUNG wire#w2
   RUNG wire#w1
      { S7_Templates := "SrcType := Int" } EQ_Contact(in1 := "DB611".StepDelay."Noof StepsPv", in2 := 8)
   END_RUNG wire#w2
   RUNG wire#w1
      { S7_Templates := "SrcType := Int" } EQ_Contact(in1 := "DB611".StepDelay."Noof StepsPv", in2 := 9)
   END_RUNG wire#w2
   RUNG wire#w1
      { S7_Templates := "SrcType := Int" } EQ_Contact(in1 := "DB611".StepDelay."Noof StepsPv", in2 := 10)
   END_RUNG wire#w2
   RUNG wire#w1
      { S7_Templates := "SrcType := Int" } EQ_Contact(in1 := "DB611".StepDelay."Noof StepsPv", in2 := 11)
   END_RUNG wire#w2
   RUNG wire#w1
      { S7_Templates := "SrcType := Int" } EQ_Contact(in1 := "DB611".StepDelay."Noof StepsPv", in2 := 16)
   END_RUNG wire#w2
   RUNG wire#w1
      { S7_Templates := "SrcType := Int" } EQ_Contact(in1 := "DB615".CurrentStep, in2 := 9)
   END_RUNG wire#w2
   RUNG wire#w1
      { S7_Templates := "SrcType := Int" } EQ_Contact(in1 := "DB615".CurrentStep, in2 := 10)
   END_RUNG wire#w2
   RUNG wire#w1
      { S7_Templates := "SrcType := Int" } EQ_Contact(in1 := "DB615".CurrentStep, in2 := 11)
   END_RUNG wire#w2
   RUNG wire#w1
      { S7_Templates := "SrcType := Int" } EQ_Contact(in1 := "DB615".CurrentStep, in2 := 15)
   END_RUNG wire#w2
   RUNG wire#w1
      { S7_Templates := "SrcType := Int" } EQ_Contact(in1 := "DB615".CurrentStep, in2 := 16)
   END_RUNG wire#w2
   RUNG wire#w1
      { S7_Templates := "SrcType := Int" } EQ_Contact(in1 := "DB611".StepDelay."Noof StepsPv", in2 := 15)
   END_RUNG wire#w2
   RUNG wire#w1
      { S7_Templates := "SrcType := Int" } EQ_Contact(in1 := "DB611".StepDelay."Noof StepsPv", in2 := 12)
      wire#w3
      { S7_Templates := "[card := 2, value_type := Real]" } MIN(in1 := "AiDb".Ai11.ActValue, in2 := "AiDb".Ai13.ActValue, out => "DB615".ApActPressure)
   END_RUNG
   RUNG wire#w1
      { S7_Templates := "SrcType := Int" } EQ_Contact(in1 := "DB611".StepDelay."Noof StepsPv", in2 := 13)
   END_RUNG wire#w3
   RUNG wire#w1
      { S7_Templates := "SrcType := Int" } EQ_Contact(in1 := "DB611".StepDelay."Noof StepsPv", in2 := 14)
      wire#w4
      { S7_Templates := "[card := 3, value_type := Real]" } MIN(in1 := "AiDb".Ai11.ActValue, in2 := "AiDb".Ai13.ActValue, in3 := "AiDb".Ai14.ActValue, out => "DB615".ApActPressure)
   END_RUNG
   RUNG wire#w1
      { S7_Templates := "SrcType := Int" } EQ_Contact(in1 := "DB611".StepDelay."Noof StepsPv", in2 := 17)
   END_RUNG wire#w4
   RUNG wire#w1
      { S7_Templates := "SrcType := Int" } EQ_Contact(in1 := "DB611".StepDelay."Noof StepsPv", in2 := 6)
      Move(in := "AiDb".Ai12.ActValue, out1 => "DB615".ApActPressure)
   END_RUNG
   // the same network as SCL:
   #_w1 := "AlwaysTRUE" AND "DB615".Selected;
   IF #_w1 AND (("DB611".StepDelay."Noof StepsPv" <= 5) OR ("DB611".StepDelay."Noof StepsPv" = 7) OR ("DB611".StepDelay."Noof StepsPv" = 8) OR ("DB611".StepDelay."Noof StepsPv" = 9) OR ("DB611".StepDelay."Noof StepsPv" = 10) OR ("DB611".StepDelay."Noof StepsPv" = 11) OR ("DB611".StepDelay."Noof StepsPv" = 16) OR ("DB615".CurrentStep = 9) OR ("DB615".CurrentStep = 10) OR ("DB615".CurrentStep = 11) OR ("DB615".CurrentStep = 15) OR ("DB615".CurrentStep = 16) OR ("DB611".StepDelay."Noof StepsPv" = 15)) THEN
       "DB615".ApActPressure := "AiDb".Ai11.ActValue;
   END_IF;
   IF #_w1 AND (("DB611".StepDelay."Noof StepsPv" = 12) OR ("DB611".StepDelay."Noof StepsPv" = 13)) THEN
       "DB615".ApActPressure := MIN(IN1 := "AiDb".Ai11.ActValue, IN2 := "AiDb".Ai13.ActValue);
   END_IF;
   IF #_w1 AND (("DB611".StepDelay."Noof StepsPv" = 14) OR ("DB611".StepDelay."Noof StepsPv" = 17)) THEN
       "DB615".ApActPressure := MIN(IN1 := "AiDb".Ai11.ActValue, IN2 := "AiDb".Ai13.ActValue, IN3 := "AiDb".Ai14.ActValue);
   END_IF;
   IF #_w1 AND ("DB611".StepDelay."Noof StepsPv" = 6) THEN
       "DB615".ApActPressure := "AiDb".Ai12.ActValue;
   END_IF;
END_REGION
END_FUNCTION

FUNCTION "CipEvents" : Void   // FC2, LAD
{ S7_Optimized_Access := 'TRUE' }
// stored: SetENOAutomatically false
   VAR_TEMP   // added for the SCL form of the ladder/FBD networks
      _w1 : Bool;
      _w2 : Bool;
      _w3 : Bool;
      _w4 : Bool;
      _w5 : Bool;
      _w6 : Bool;
      _w7 : Bool;
      _w8 : Bool;
      _w9 : Bool;
      _w10 : Bool;
      _w11 : Bool;
      _w12 : Bool;
      _w13 : Bool;
      _w14 : Bool;
      _w15 : Bool;
      _w16 : Bool;
      _w17 : Bool;
      _w18 : Bool;
      _w19 : Bool;
      _w20 : Bool;
      _w21 : Bool;
      _w22 : Bool;
      _w23 : Bool;
      _w24 : Bool;
      _w25 : Bool;
      _w26 : Bool;
      _w27 : Bool;
      _w28 : Bool;
      _w29 : Bool;
      _w30 : Bool;
      _w31 : Bool;
      _w32 : Bool;
      _w33 : Bool;
      _w34 : Bool;
      _w35 : Bool;
      _w36 : Bool;
      _w37 : Bool;
      _w38 : Bool;
      _w39 : Bool;
      _w40 : Bool;
   END_VAR
BEGIN

REGION Network 1: ****************D500****************
END_REGION

REGION Network 2: Events And Line Print
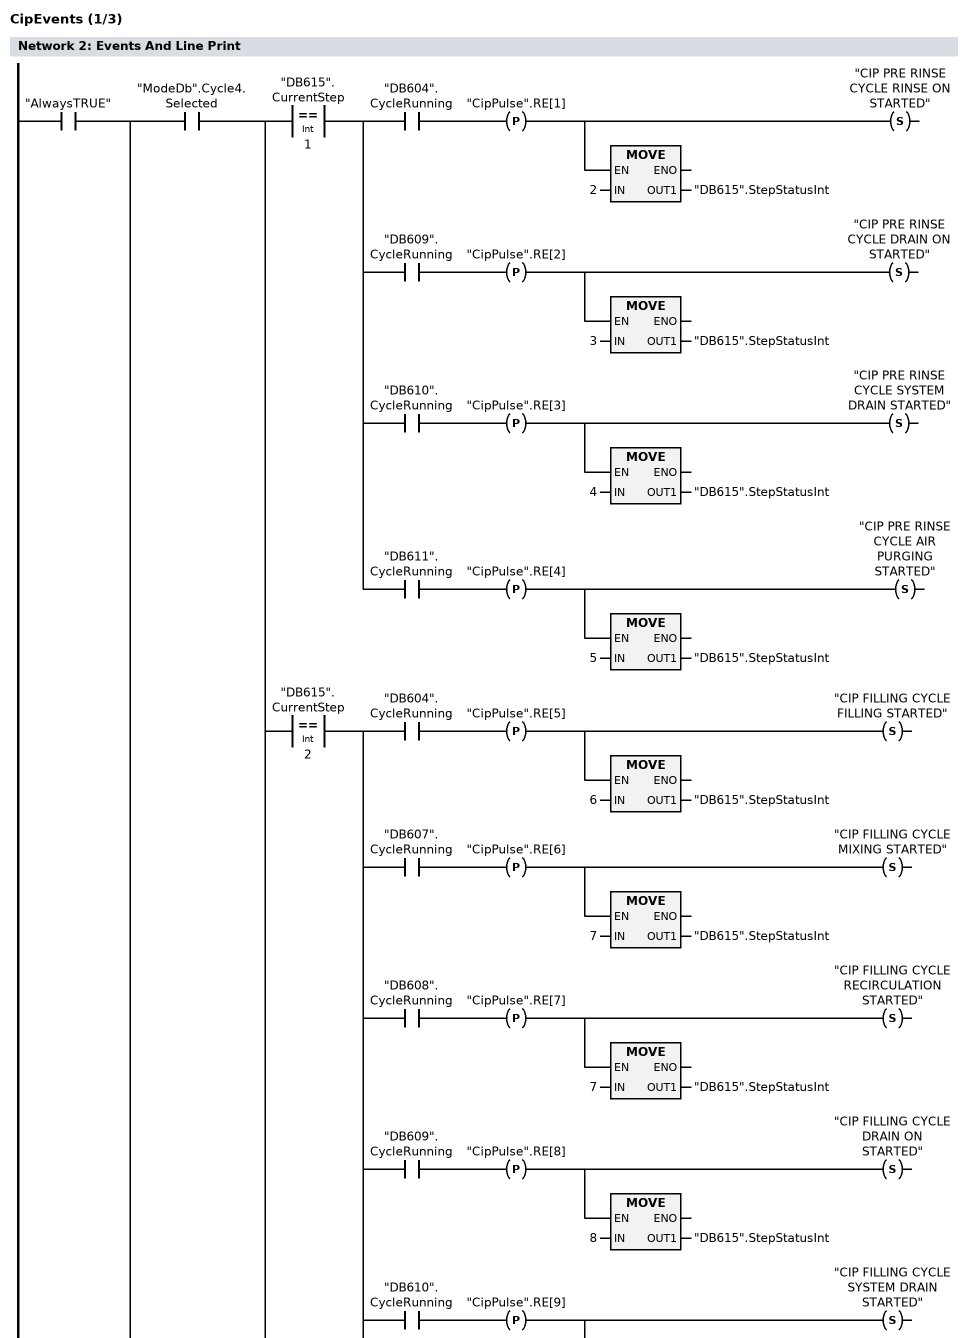
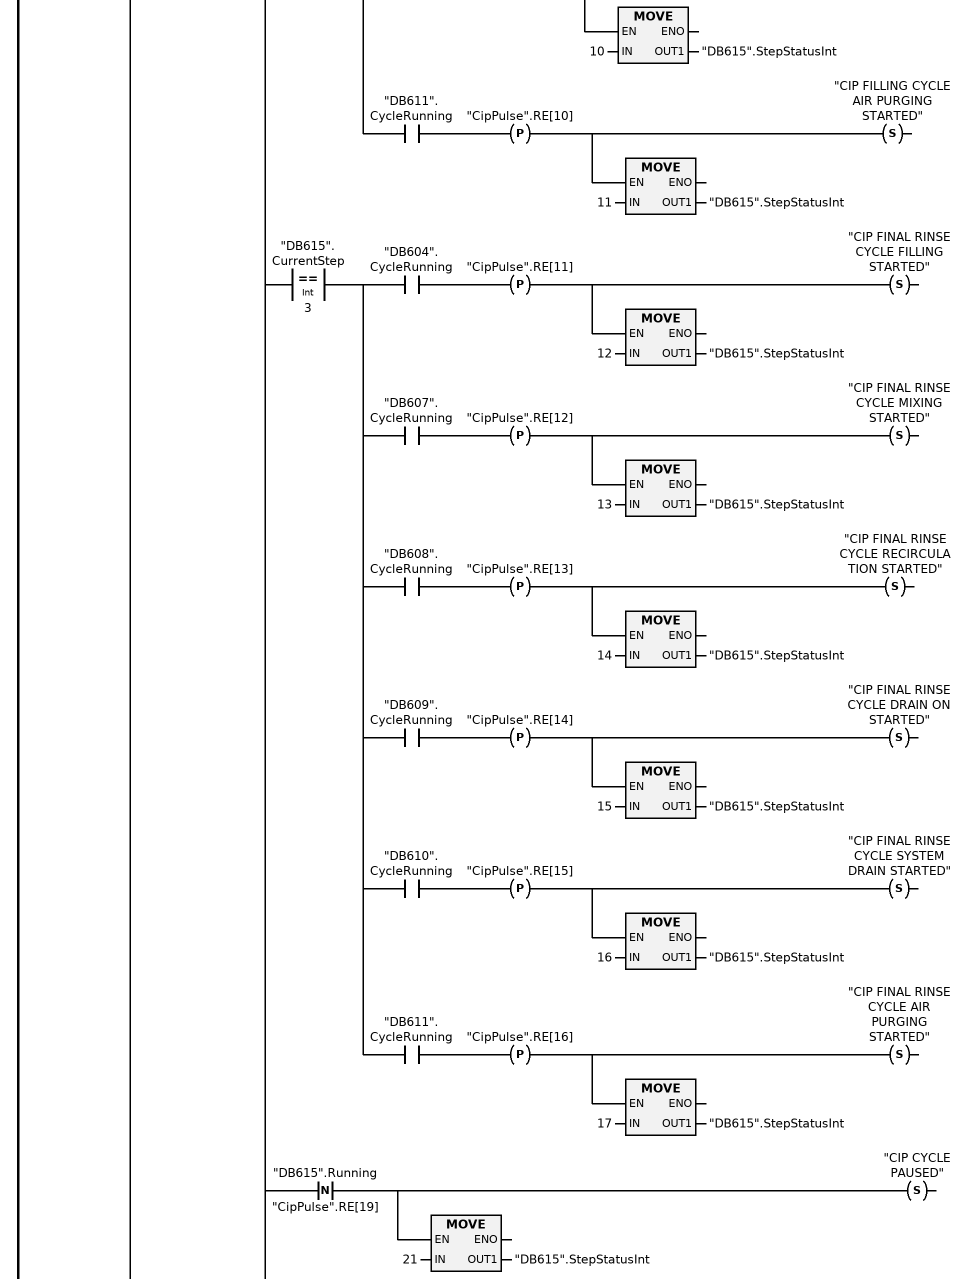
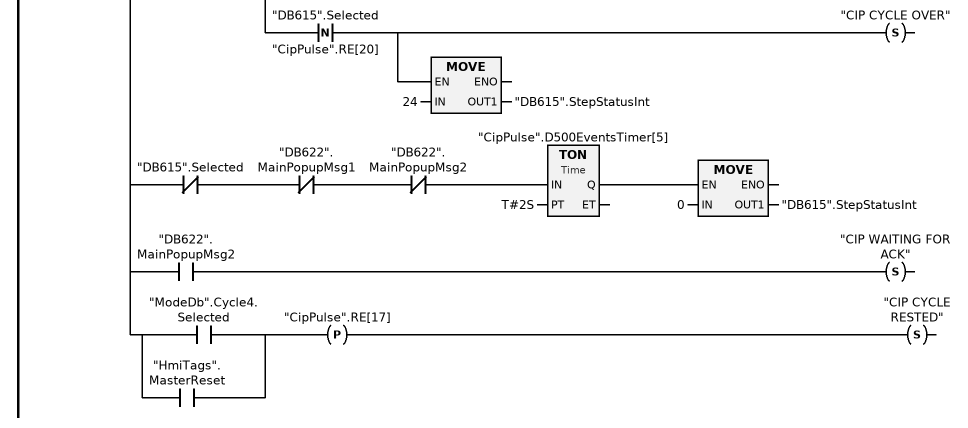
   RUNG wire#powerrail
      Contact( "AlwaysTRUE" )
      wire#w1
      Contact( "ModeDb".Cycle4.Selected )
      wire#w2
      { S7_Templates := "SrcType := Int" } EQ_Contact(in1 := "DB615".CurrentStep, in2 := 1)
      wire#w3
      Contact( "DB604".CycleRunning )
      P_Trig( "CipPulse".RE[1] )
      wire#w4
      S_Coil( "CIP PRE RINSE CYCLE RINSE ON STARTED" )
   END_RUNG
   RUNG wire#w4
      Move(in := 2, out1 => "DB615".StepStatusInt)
   END_RUNG
   RUNG wire#w3
      Contact( "DB609".CycleRunning )
      P_Trig( "CipPulse".RE[2] )
      wire#w5
      S_Coil( "CIP PRE RINSE CYCLE DRAIN ON STARTED" )
   END_RUNG
   RUNG wire#w5
      Move(in := 3, out1 => "DB615".StepStatusInt)
   END_RUNG
   RUNG wire#w3
      Contact( "DB610".CycleRunning )
      P_Trig( "CipPulse".RE[3] )
      wire#w6
      S_Coil( "CIP PRE RINSE CYCLE SYSTEM DRAIN STARTED" )
   END_RUNG
   RUNG wire#w6
      Move(in := 4, out1 => "DB615".StepStatusInt)
   END_RUNG
   RUNG wire#w3
      Contact( "DB611".CycleRunning )
      P_Trig( "CipPulse".RE[4] )
      wire#w7
      S_Coil( "CIP PRE RINSE CYCLE AIR PURGING STARTED" )
   END_RUNG
   RUNG wire#w7
      Move(in := 5, out1 => "DB615".StepStatusInt)
   END_RUNG
   RUNG wire#w2
      { S7_Templates := "SrcType := Int" } EQ_Contact(in1 := "DB615".CurrentStep, in2 := 2)
      wire#w8
      Contact( "DB604".CycleRunning )
      P_Trig( "CipPulse".RE[5] )
      wire#w9
      S_Coil( "CIP FILLING CYCLE FILLING STARTED" )
   END_RUNG
   RUNG wire#w9
      Move(in := 6, out1 => "DB615".StepStatusInt)
   END_RUNG
   RUNG wire#w8
      Contact( "DB607".CycleRunning )
      P_Trig( "CipPulse".RE[6] )
      wire#w10
      S_Coil( "CIP FILLING CYCLE MIXING STARTED" )
   END_RUNG
   RUNG wire#w10
      Move(in := 7, out1 => "DB615".StepStatusInt)
   END_RUNG
   RUNG wire#w8
      Contact( "DB608".CycleRunning )
      P_Trig( "CipPulse".RE[7] )
      wire#w11
      S_Coil( "CIP FILLING CYCLE RECIRCULATION STARTED" )
   END_RUNG
   RUNG wire#w11
      Move(in := 7, out1 => "DB615".StepStatusInt)
   END_RUNG
   RUNG wire#w8
      Contact( "DB609".CycleRunning )
      P_Trig( "CipPulse".RE[8] )
      wire#w12
      S_Coil( "CIP FILLING CYCLE DRAIN ON STARTED" )
   END_RUNG
   RUNG wire#w12
      Move(in := 8, out1 => "DB615".StepStatusInt)
   END_RUNG
   RUNG wire#w8
      Contact( "DB610".CycleRunning )
      P_Trig( "CipPulse".RE[9] )
      wire#w13
      S_Coil( "CIP FILLING CYCLE SYSTEM DRAIN STARTED" )
   END_RUNG
   RUNG wire#w13
      Move(in := 10, out1 => "DB615".StepStatusInt)
   END_RUNG
   RUNG wire#w8
      Contact( "DB611".CycleRunning )
      P_Trig( "CipPulse".RE[10] )
      wire#w14
      S_Coil( "CIP FILLING CYCLE AIR PURGING STARTED" )
   END_RUNG
   RUNG wire#w14
      Move(in := 11, out1 => "DB615".StepStatusInt)
   END_RUNG
   RUNG wire#w2
      { S7_Templates := "SrcType := Int" } EQ_Contact(in1 := "DB615".CurrentStep, in2 := 3)
      wire#w15
      Contact( "DB604".CycleRunning )
      P_Trig( "CipPulse".RE[11] )
      wire#w16
      S_Coil( "CIP FINAL RINSE CYCLE FILLING STARTED" )
   END_RUNG
   RUNG wire#w16
      Move(in := 12, out1 => "DB615".StepStatusInt)
   END_RUNG
   RUNG wire#w15
      Contact( "DB607".CycleRunning )
      P_Trig( "CipPulse".RE[12] )
      wire#w17
      S_Coil( "CIP FINAL RINSE CYCLE MIXING STARTED" )
   END_RUNG
   RUNG wire#w17
      Move(in := 13, out1 => "DB615".StepStatusInt)
   END_RUNG
   RUNG wire#w15
      Contact( "DB608".CycleRunning )
      P_Trig( "CipPulse".RE[13] )
      wire#w18
      S_Coil( "CIP FINAL RINSE CYCLE RECIRCULATION STARTED" )
   END_RUNG
   RUNG wire#w18
      Move(in := 14, out1 => "DB615".StepStatusInt)
   END_RUNG
   RUNG wire#w15
      Contact( "DB609".CycleRunning )
      P_Trig( "CipPulse".RE[14] )
      wire#w19
      S_Coil( "CIP FINAL RINSE CYCLE DRAIN ON STARTED" )
   END_RUNG
   RUNG wire#w19
      Move(in := 15, out1 => "DB615".StepStatusInt)
   END_RUNG
   RUNG wire#w15
      Contact( "DB610".CycleRunning )
      P_Trig( "CipPulse".RE[15] )
      wire#w20
      S_Coil( "CIP FINAL RINSE CYCLE SYSTEM DRAIN STARTED" )
   END_RUNG
   RUNG wire#w20
      Move(in := 16, out1 => "DB615".StepStatusInt)
   END_RUNG
   RUNG wire#w15
      Contact( "DB611".CycleRunning )
      P_Trig( "CipPulse".RE[16] )
      wire#w21
      S_Coil( "CIP FINAL RINSE CYCLE AIR PURGING STARTED" )
   END_RUNG
   RUNG wire#w21
      Move(in := 17, out1 => "DB615".StepStatusInt)
   END_RUNG
   RUNG wire#w2
      N_Contact(operand := "DB615".Running, bit := "CipPulse".RE[19])
      wire#w22
      S_Coil( "CIP CYCLE PAUSED" )
   END_RUNG
   RUNG wire#w22
      Move(in := 21, out1 => "DB615".StepStatusInt)
   END_RUNG
   RUNG wire#w2
      N_Contact(operand := "DB615".Selected, bit := "CipPulse".RE[20])
      wire#w23
      S_Coil( "CIP CYCLE OVER" )
   END_RUNG
   RUNG wire#w23
      Move(in := 24, out1 => "DB615".StepStatusInt)
   END_RUNG
   RUNG wire#w1
      I_Contact( "DB615".Selected )
      I_Contact( "DB622".MainPopupMsg1 )
      I_Contact( "DB622".MainPopupMsg2 )
      { S7_Templates := "time_type := Time" } "CipPulse".D500EventsTimer[5].TON(pt := T#2S, et =>)
      Move(in := 0, out1 => "DB615".StepStatusInt)
   END_RUNG
   RUNG wire#w1
      Contact( "DB622".MainPopupMsg2 )
      S_Coil( "CIP WAITING FOR ACK" )
   END_RUNG
   RUNG wire#w1
      Contact( "ModeDb".Cycle4.Selected )
      wire#w24
      P_Trig( "CipPulse".RE[17] )
      S_Coil( "CIP CYCLE RESTED" )
   END_RUNG
   RUNG wire#w1
      Contact( "HmiTags".MasterReset )
   END_RUNG wire#w24
   // the same network as SCL:
   #_w1 := "AlwaysTRUE" AND "ModeDb".Cycle4.Selected;
   #_w2 := #_w1 AND ("DB615".CurrentStep = 1);
   #_w3 := #_w2 AND "DB604".CycleRunning;
   #_w4 := #_w3 AND NOT "CipPulse".RE[1];   // rising edge
   "CipPulse".RE[1] := #_w3;
   IF #_w4 THEN
       "CIP PRE RINSE CYCLE RINSE ON STARTED" := TRUE;
       "DB615".StepStatusInt := 2;
   END_IF;
   #_w5 := #_w2 AND "DB609".CycleRunning;
   #_w6 := #_w5 AND NOT "CipPulse".RE[2];   // rising edge
   "CipPulse".RE[2] := #_w5;
   IF #_w6 THEN
       "CIP PRE RINSE CYCLE DRAIN ON STARTED" := TRUE;
       "DB615".StepStatusInt := 3;
   END_IF;
   #_w7 := #_w2 AND "DB610".CycleRunning;
   #_w8 := #_w7 AND NOT "CipPulse".RE[3];   // rising edge
   "CipPulse".RE[3] := #_w7;
   IF #_w8 THEN
       "CIP PRE RINSE CYCLE SYSTEM DRAIN STARTED" := TRUE;
       "DB615".StepStatusInt := 4;
   END_IF;
   #_w9 := #_w2 AND "DB611".CycleRunning;
   #_w10 := #_w9 AND NOT "CipPulse".RE[4];   // rising edge
   "CipPulse".RE[4] := #_w9;
   IF #_w10 THEN
       "CIP PRE RINSE CYCLE AIR PURGING STARTED" := TRUE;
       "DB615".StepStatusInt := 5;
   END_IF;
   #_w11 := #_w1 AND ("DB615".CurrentStep = 2);
   #_w12 := #_w11 AND "DB604".CycleRunning;
   #_w13 := #_w12 AND NOT "CipPulse".RE[5];   // rising edge
   "CipPulse".RE[5] := #_w12;
   IF #_w13 THEN
       "CIP FILLING CYCLE FILLING STARTED" := TRUE;
       "DB615".StepStatusInt := 6;
   END_IF;
   #_w14 := #_w11 AND "DB607".CycleRunning;
   #_w15 := #_w14 AND NOT "CipPulse".RE[6];   // rising edge
   "CipPulse".RE[6] := #_w14;
   IF #_w15 THEN
       "CIP FILLING CYCLE MIXING STARTED" := TRUE;
       "DB615".StepStatusInt := 7;
   END_IF;
   #_w16 := #_w11 AND "DB608".CycleRunning;
   #_w17 := #_w16 AND NOT "CipPulse".RE[7];   // rising edge
   "CipPulse".RE[7] := #_w16;
   IF #_w17 THEN
       "CIP FILLING CYCLE RECIRCULATION STARTED" := TRUE;
       "DB615".StepStatusInt := 7;
   END_IF;
   #_w18 := #_w11 AND "DB609".CycleRunning;
   #_w19 := #_w18 AND NOT "CipPulse".RE[8];   // rising edge
   "CipPulse".RE[8] := #_w18;
   IF #_w19 THEN
       "CIP FILLING CYCLE DRAIN ON STARTED" := TRUE;
       "DB615".StepStatusInt := 8;
   END_IF;
   #_w20 := #_w11 AND "DB610".CycleRunning;
   #_w21 := #_w20 AND NOT "CipPulse".RE[9];   // rising edge
   "CipPulse".RE[9] := #_w20;
   IF #_w21 THEN
       "CIP FILLING CYCLE SYSTEM DRAIN STARTED" := TRUE;
       "DB615".StepStatusInt := 10;
   END_IF;
   #_w22 := #_w11 AND "DB611".CycleRunning;
   #_w23 := #_w22 AND NOT "CipPulse".RE[10];   // rising edge
   "CipPulse".RE[10] := #_w22;
   IF #_w23 THEN
       "CIP FILLING CYCLE AIR PURGING STARTED" := TRUE;
       "DB615".StepStatusInt := 11;
   END_IF;
   #_w24 := #_w1 AND ("DB615".CurrentStep = 3);
   #_w25 := #_w24 AND "DB604".CycleRunning;
   #_w26 := #_w25 AND NOT "CipPulse".RE[11];   // rising edge
   "CipPulse".RE[11] := #_w25;
   IF #_w26 THEN
       "CIP FINAL RINSE CYCLE FILLING STARTED" := TRUE;
       "DB615".StepStatusInt := 12;
   END_IF;
   #_w27 := #_w24 AND "DB607".CycleRunning;
   #_w28 := #_w27 AND NOT "CipPulse".RE[12];   // rising edge
   "CipPulse".RE[12] := #_w27;
   IF #_w28 THEN
       "CIP FINAL RINSE CYCLE MIXING STARTED" := TRUE;
       "DB615".StepStatusInt := 13;
   END_IF;
   #_w29 := #_w24 AND "DB608".CycleRunning;
   #_w30 := #_w29 AND NOT "CipPulse".RE[13];   // rising edge
   "CipPulse".RE[13] := #_w29;
   IF #_w30 THEN
       "CIP FINAL RINSE CYCLE RECIRCULATION STARTED" := TRUE;
       "DB615".StepStatusInt := 14;
   END_IF;
   #_w31 := #_w24 AND "DB609".CycleRunning;
   #_w32 := #_w31 AND NOT "CipPulse".RE[14];   // rising edge
   "CipPulse".RE[14] := #_w31;
   IF #_w32 THEN
       "CIP FINAL RINSE CYCLE DRAIN ON STARTED" := TRUE;
       "DB615".StepStatusInt := 15;
   END_IF;
   #_w33 := #_w24 AND "DB610".CycleRunning;
   #_w34 := #_w33 AND NOT "CipPulse".RE[15];   // rising edge
   "CipPulse".RE[15] := #_w33;
   IF #_w34 THEN
       "CIP FINAL RINSE CYCLE SYSTEM DRAIN STARTED" := TRUE;
       "DB615".StepStatusInt := 16;
   END_IF;
   #_w35 := #_w24 AND "DB611".CycleRunning;
   #_w36 := #_w35 AND NOT "CipPulse".RE[16];   // rising edge
   "CipPulse".RE[16] := #_w35;
   IF #_w36 THEN
       "CIP FINAL RINSE CYCLE AIR PURGING STARTED" := TRUE;
       "DB615".StepStatusInt := 17;
   END_IF;
   #_w37 := #_w1 AND NOT "DB615".Running AND "CipPulse".RE[19];   // falling edge of "DB615".Running
   "CipPulse".RE[19] := "DB615".Running;
   IF #_w37 THEN
       "CIP CYCLE PAUSED" := TRUE;
       "DB615".StepStatusInt := 21;
   END_IF;
   #_w38 := #_w1 AND NOT "DB615".Selected AND "CipPulse".RE[20];   // falling edge of "DB615".Selected
   "CipPulse".RE[20] := "DB615".Selected;
   IF #_w38 THEN
       "CIP CYCLE OVER" := TRUE;
       "DB615".StepStatusInt := 24;
   END_IF;
   "CipPulse".D500EventsTimer[5].TON(IN := "AlwaysTRUE" AND NOT "DB615".Selected AND NOT "DB622".MainPopupMsg1 AND NOT "DB622".MainPopupMsg2,
                           PT := T#2S);
   IF "CipPulse".D500EventsTimer[5].Q THEN "DB615".StepStatusInt := 0; END_IF;
   IF "AlwaysTRUE" AND "DB622".MainPopupMsg2 THEN "CIP WAITING FOR ACK" := TRUE; END_IF;
   #_w39 := "AlwaysTRUE" AND ("ModeDb".Cycle4.Selected OR "HmiTags".MasterReset);
   #_w40 := #_w39 AND NOT "CipPulse".RE[17];   // rising edge
   "CipPulse".RE[17] := #_w39;
   IF #_w40 THEN "CIP CYCLE RESTED" := TRUE; END_IF;
END_REGION

REGION Network 3: PRE RINSE
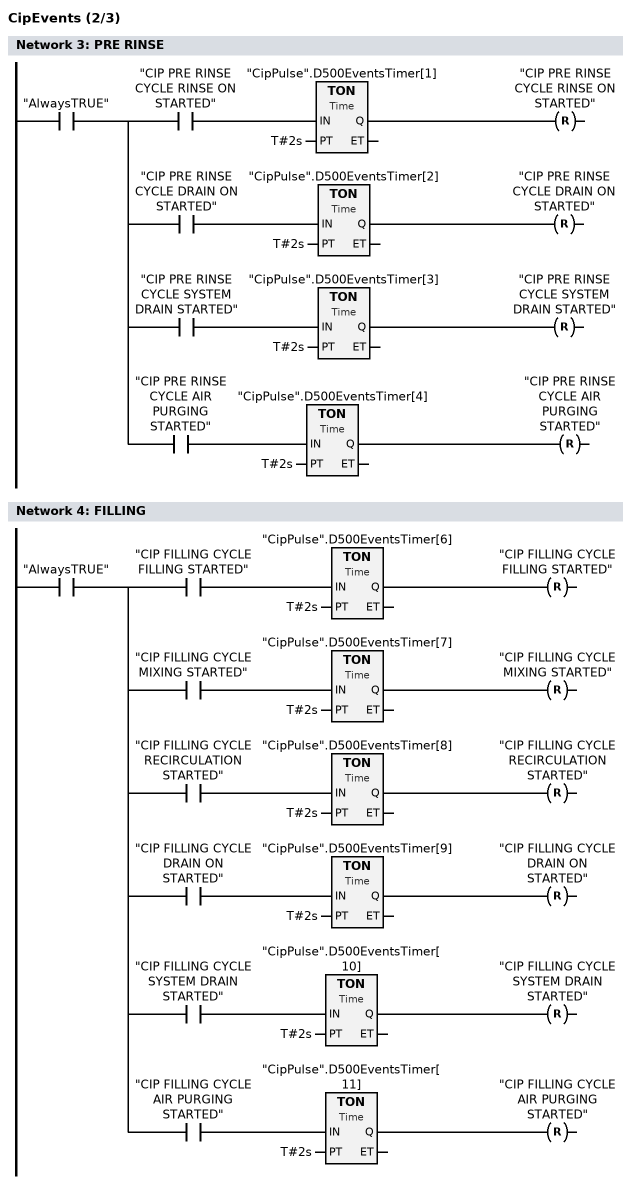
   RUNG wire#powerrail
      Contact( "AlwaysTRUE" )
      wire#w1
      Contact( "CIP PRE RINSE CYCLE RINSE ON STARTED" )
      { S7_Templates := "time_type := Time" } "CipPulse".D500EventsTimer[1].TON(pt := T#2s, et =>)
      R_Coil( "CIP PRE RINSE CYCLE RINSE ON STARTED" )
   END_RUNG
   RUNG wire#w1
      Contact( "CIP PRE RINSE CYCLE DRAIN ON STARTED" )
      { S7_Templates := "time_type := Time" } "CipPulse".D500EventsTimer[2].TON(pt := T#2s, et =>)
      R_Coil( "CIP PRE RINSE CYCLE DRAIN ON STARTED" )
   END_RUNG
   RUNG wire#w1
      Contact( "CIP PRE RINSE CYCLE SYSTEM DRAIN STARTED" )
      { S7_Templates := "time_type := Time" } "CipPulse".D500EventsTimer[3].TON(pt := T#2s, et =>)
      R_Coil( "CIP PRE RINSE CYCLE SYSTEM DRAIN STARTED" )
   END_RUNG
   RUNG wire#w1
      Contact( "CIP PRE RINSE CYCLE AIR PURGING STARTED" )
      { S7_Templates := "time_type := Time" } "CipPulse".D500EventsTimer[4].TON(pt := T#2s, et =>)
      R_Coil( "CIP PRE RINSE CYCLE AIR PURGING STARTED" )
   END_RUNG
   // the same network as SCL:
   "CipPulse".D500EventsTimer[1].TON(IN := "AlwaysTRUE" AND "CIP PRE RINSE CYCLE RINSE ON STARTED", PT := T#2s);
   IF "CipPulse".D500EventsTimer[1].Q THEN "CIP PRE RINSE CYCLE RINSE ON STARTED" := FALSE; END_IF;
   "CipPulse".D500EventsTimer[2].TON(IN := "AlwaysTRUE" AND "CIP PRE RINSE CYCLE DRAIN ON STARTED", PT := T#2s);
   IF "CipPulse".D500EventsTimer[2].Q THEN "CIP PRE RINSE CYCLE DRAIN ON STARTED" := FALSE; END_IF;
   "CipPulse".D500EventsTimer[3].TON(IN := "AlwaysTRUE" AND "CIP PRE RINSE CYCLE SYSTEM DRAIN STARTED",
                           PT := T#2s);
   IF "CipPulse".D500EventsTimer[3].Q THEN "CIP PRE RINSE CYCLE SYSTEM DRAIN STARTED" := FALSE; END_IF;
   "CipPulse".D500EventsTimer[4].TON(IN := "AlwaysTRUE" AND "CIP PRE RINSE CYCLE AIR PURGING STARTED",
                           PT := T#2s);
   IF "CipPulse".D500EventsTimer[4].Q THEN "CIP PRE RINSE CYCLE AIR PURGING STARTED" := FALSE; END_IF;
END_REGION

REGION Network 4: FILLING
   RUNG wire#powerrail
      Contact( "AlwaysTRUE" )
      wire#w1
      Contact( "CIP FILLING CYCLE FILLING STARTED" )
      { S7_Templates := "time_type := Time" } "CipPulse".D500EventsTimer[6].TON(pt := T#2s, et =>)
      R_Coil( "CIP FILLING CYCLE FILLING STARTED" )
   END_RUNG
   RUNG wire#w1
      Contact( "CIP FILLING CYCLE MIXING STARTED" )
      { S7_Templates := "time_type := Time" } "CipPulse".D500EventsTimer[7].TON(pt := T#2s, et =>)
      R_Coil( "CIP FILLING CYCLE MIXING STARTED" )
   END_RUNG
   RUNG wire#w1
      Contact( "CIP FILLING CYCLE RECIRCULATION STARTED" )
      { S7_Templates := "time_type := Time" } "CipPulse".D500EventsTimer[8].TON(pt := T#2s, et =>)
      R_Coil( "CIP FILLING CYCLE RECIRCULATION STARTED" )
   END_RUNG
   RUNG wire#w1
      Contact( "CIP FILLING CYCLE DRAIN ON STARTED" )
      { S7_Templates := "time_type := Time" } "CipPulse".D500EventsTimer[9].TON(pt := T#2s, et =>)
      R_Coil( "CIP FILLING CYCLE DRAIN ON STARTED" )
   END_RUNG
   RUNG wire#w1
      Contact( "CIP FILLING CYCLE SYSTEM DRAIN STARTED" )
      { S7_Templates := "time_type := Time" } "CipPulse".D500EventsTimer[10].TON(pt := T#2s, et =>)
      R_Coil( "CIP FILLING CYCLE SYSTEM DRAIN STARTED" )
   END_RUNG
   RUNG wire#w1
      Contact( "CIP FILLING CYCLE AIR PURGING STARTED" )
      { S7_Templates := "time_type := Time" } "CipPulse".D500EventsTimer[11].TON(pt := T#2s, et =>)
      R_Coil( "CIP FILLING CYCLE AIR PURGING STARTED" )
   END_RUNG
   // the same network as SCL:
   "CipPulse".D500EventsTimer[6].TON(IN := "AlwaysTRUE" AND "CIP FILLING CYCLE FILLING STARTED", PT := T#2s);
   IF "CipPulse".D500EventsTimer[6].Q THEN "CIP FILLING CYCLE FILLING STARTED" := FALSE; END_IF;
   "CipPulse".D500EventsTimer[7].TON(IN := "AlwaysTRUE" AND "CIP FILLING CYCLE MIXING STARTED", PT := T#2s);
   IF "CipPulse".D500EventsTimer[7].Q THEN "CIP FILLING CYCLE MIXING STARTED" := FALSE; END_IF;
   "CipPulse".D500EventsTimer[8].TON(IN := "AlwaysTRUE" AND "CIP FILLING CYCLE RECIRCULATION STARTED",
                           PT := T#2s);
   IF "CipPulse".D500EventsTimer[8].Q THEN "CIP FILLING CYCLE RECIRCULATION STARTED" := FALSE; END_IF;
   "CipPulse".D500EventsTimer[9].TON(IN := "AlwaysTRUE" AND "CIP FILLING CYCLE DRAIN ON STARTED", PT := T#2s);
   IF "CipPulse".D500EventsTimer[9].Q THEN "CIP FILLING CYCLE DRAIN ON STARTED" := FALSE; END_IF;
   "CipPulse".D500EventsTimer[10].TON(IN := "AlwaysTRUE" AND "CIP FILLING CYCLE SYSTEM DRAIN STARTED",
                           PT := T#2s);
   IF "CipPulse".D500EventsTimer[10].Q THEN "CIP FILLING CYCLE SYSTEM DRAIN STARTED" := FALSE; END_IF;
   "CipPulse".D500EventsTimer[11].TON(IN := "AlwaysTRUE" AND "CIP FILLING CYCLE AIR PURGING STARTED",
                           PT := T#2s);
   IF "CipPulse".D500EventsTimer[11].Q THEN "CIP FILLING CYCLE AIR PURGING STARTED" := FALSE; END_IF;
END_REGION

REGION Network 5: FINAL RINSE
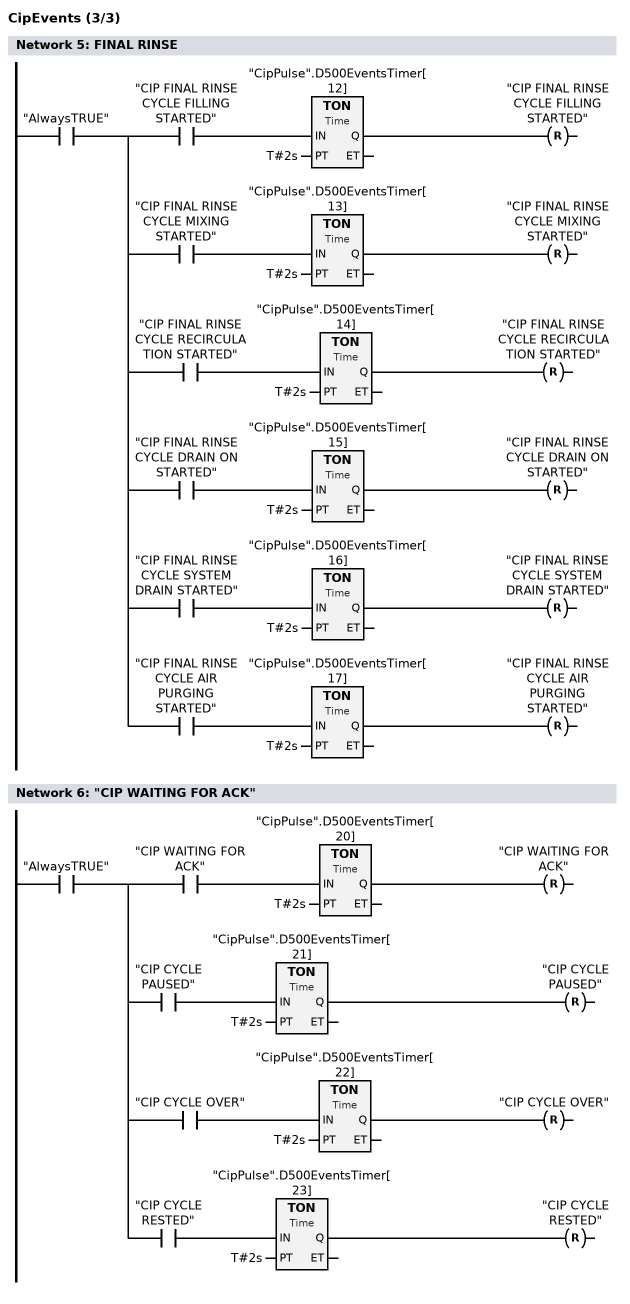
   RUNG wire#powerrail
      Contact( "AlwaysTRUE" )
      wire#w1
      Contact( "CIP FINAL RINSE CYCLE FILLING STARTED" )
      { S7_Templates := "time_type := Time" } "CipPulse".D500EventsTimer[12].TON(pt := T#2s, et =>)
      R_Coil( "CIP FINAL RINSE CYCLE FILLING STARTED" )
   END_RUNG
   RUNG wire#w1
      Contact( "CIP FINAL RINSE CYCLE MIXING STARTED" )
      { S7_Templates := "time_type := Time" } "CipPulse".D500EventsTimer[13].TON(pt := T#2s, et =>)
      R_Coil( "CIP FINAL RINSE CYCLE MIXING STARTED" )
   END_RUNG
   RUNG wire#w1
      Contact( "CIP FINAL RINSE CYCLE RECIRCULATION STARTED" )
      { S7_Templates := "time_type := Time" } "CipPulse".D500EventsTimer[14].TON(pt := T#2s, et =>)
      R_Coil( "CIP FINAL RINSE CYCLE RECIRCULATION STARTED" )
   END_RUNG
   RUNG wire#w1
      Contact( "CIP FINAL RINSE CYCLE DRAIN ON STARTED" )
      { S7_Templates := "time_type := Time" } "CipPulse".D500EventsTimer[15].TON(pt := T#2s, et =>)
      R_Coil( "CIP FINAL RINSE CYCLE DRAIN ON STARTED" )
   END_RUNG
   RUNG wire#w1
      Contact( "CIP FINAL RINSE CYCLE SYSTEM DRAIN STARTED" )
      { S7_Templates := "time_type := Time" } "CipPulse".D500EventsTimer[16].TON(pt := T#2s, et =>)
      R_Coil( "CIP FINAL RINSE CYCLE SYSTEM DRAIN STARTED" )
   END_RUNG
   RUNG wire#w1
      Contact( "CIP FINAL RINSE CYCLE AIR PURGING STARTED" )
      { S7_Templates := "time_type := Time" } "CipPulse".D500EventsTimer[17].TON(pt := T#2s, et =>)
      R_Coil( "CIP FINAL RINSE CYCLE AIR PURGING STARTED" )
   END_RUNG
   // the same network as SCL:
   "CipPulse".D500EventsTimer[12].TON(IN := "AlwaysTRUE" AND "CIP FINAL RINSE CYCLE FILLING STARTED",
                           PT := T#2s);
   IF "CipPulse".D500EventsTimer[12].Q THEN "CIP FINAL RINSE CYCLE FILLING STARTED" := FALSE; END_IF;
   "CipPulse".D500EventsTimer[13].TON(IN := "AlwaysTRUE" AND "CIP FINAL RINSE CYCLE MIXING STARTED", PT := T#2s);
   IF "CipPulse".D500EventsTimer[13].Q THEN "CIP FINAL RINSE CYCLE MIXING STARTED" := FALSE; END_IF;
   "CipPulse".D500EventsTimer[14].TON(IN := "AlwaysTRUE" AND "CIP FINAL RINSE CYCLE RECIRCULATION STARTED",
                           PT := T#2s);
   IF "CipPulse".D500EventsTimer[14].Q THEN "CIP FINAL RINSE CYCLE RECIRCULATION STARTED" := FALSE; END_IF;
   "CipPulse".D500EventsTimer[15].TON(IN := "AlwaysTRUE" AND "CIP FINAL RINSE CYCLE DRAIN ON STARTED",
                           PT := T#2s);
   IF "CipPulse".D500EventsTimer[15].Q THEN "CIP FINAL RINSE CYCLE DRAIN ON STARTED" := FALSE; END_IF;
   "CipPulse".D500EventsTimer[16].TON(IN := "AlwaysTRUE" AND "CIP FINAL RINSE CYCLE SYSTEM DRAIN STARTED",
                           PT := T#2s);
   IF "CipPulse".D500EventsTimer[16].Q THEN "CIP FINAL RINSE CYCLE SYSTEM DRAIN STARTED" := FALSE; END_IF;
   "CipPulse".D500EventsTimer[17].TON(IN := "AlwaysTRUE" AND "CIP FINAL RINSE CYCLE AIR PURGING STARTED",
                           PT := T#2s);
   IF "CipPulse".D500EventsTimer[17].Q THEN "CIP FINAL RINSE CYCLE AIR PURGING STARTED" := FALSE; END_IF;
END_REGION

REGION Network 6: "CIP WAITING FOR ACK"
   RUNG wire#powerrail
      Contact( "AlwaysTRUE" )
      wire#w1
      Contact( "CIP WAITING FOR ACK" )
      { S7_Templates := "time_type := Time" } "CipPulse".D500EventsTimer[20].TON(pt := T#2s, et =>)
      R_Coil( "CIP WAITING FOR ACK" )
   END_RUNG
   RUNG wire#w1
      Contact( "CIP CYCLE PAUSED" )
      { S7_Templates := "time_type := Time" } "CipPulse".D500EventsTimer[21].TON(pt := T#2s, et =>)
      R_Coil( "CIP CYCLE PAUSED" )
   END_RUNG
   RUNG wire#w1
      Contact( "CIP CYCLE OVER" )
      { S7_Templates := "time_type := Time" } "CipPulse".D500EventsTimer[22].TON(pt := T#2s, et =>)
      R_Coil( "CIP CYCLE OVER" )
   END_RUNG
   RUNG wire#w1
      Contact( "CIP CYCLE RESTED" )
      { S7_Templates := "time_type := Time" } "CipPulse".D500EventsTimer[23].TON(pt := T#2s, et =>)
      R_Coil( "CIP CYCLE RESTED" )
   END_RUNG
   // the same network as SCL:
   "CipPulse".D500EventsTimer[20].TON(IN := "AlwaysTRUE" AND "CIP WAITING FOR ACK", PT := T#2s);
   IF "CipPulse".D500EventsTimer[20].Q THEN "CIP WAITING FOR ACK" := FALSE; END_IF;
   "CipPulse".D500EventsTimer[21].TON(IN := "AlwaysTRUE" AND "CIP CYCLE PAUSED", PT := T#2s);
   IF "CipPulse".D500EventsTimer[21].Q THEN "CIP CYCLE PAUSED" := FALSE; END_IF;
   "CipPulse".D500EventsTimer[22].TON(IN := "AlwaysTRUE" AND "CIP CYCLE OVER", PT := T#2s);
   IF "CipPulse".D500EventsTimer[22].Q THEN "CIP CYCLE OVER" := FALSE; END_IF;
   "CipPulse".D500EventsTimer[23].TON(IN := "AlwaysTRUE" AND "CIP CYCLE RESTED", PT := T#2s);
   IF "CipPulse".D500EventsTimer[23].Q THEN "CIP CYCLE RESTED" := FALSE; END_IF;
END_REGION
END_FUNCTION

FUNCTION "FC602_Valve Logic" : Void   // FC602, LAD
{ S7_Optimized_Access := 'TRUE' }
// stored: AutoNumber false, SetENOAutomatically false
BEGIN

REGION Network 2: "CipVessel".Cv06 -------- Jv
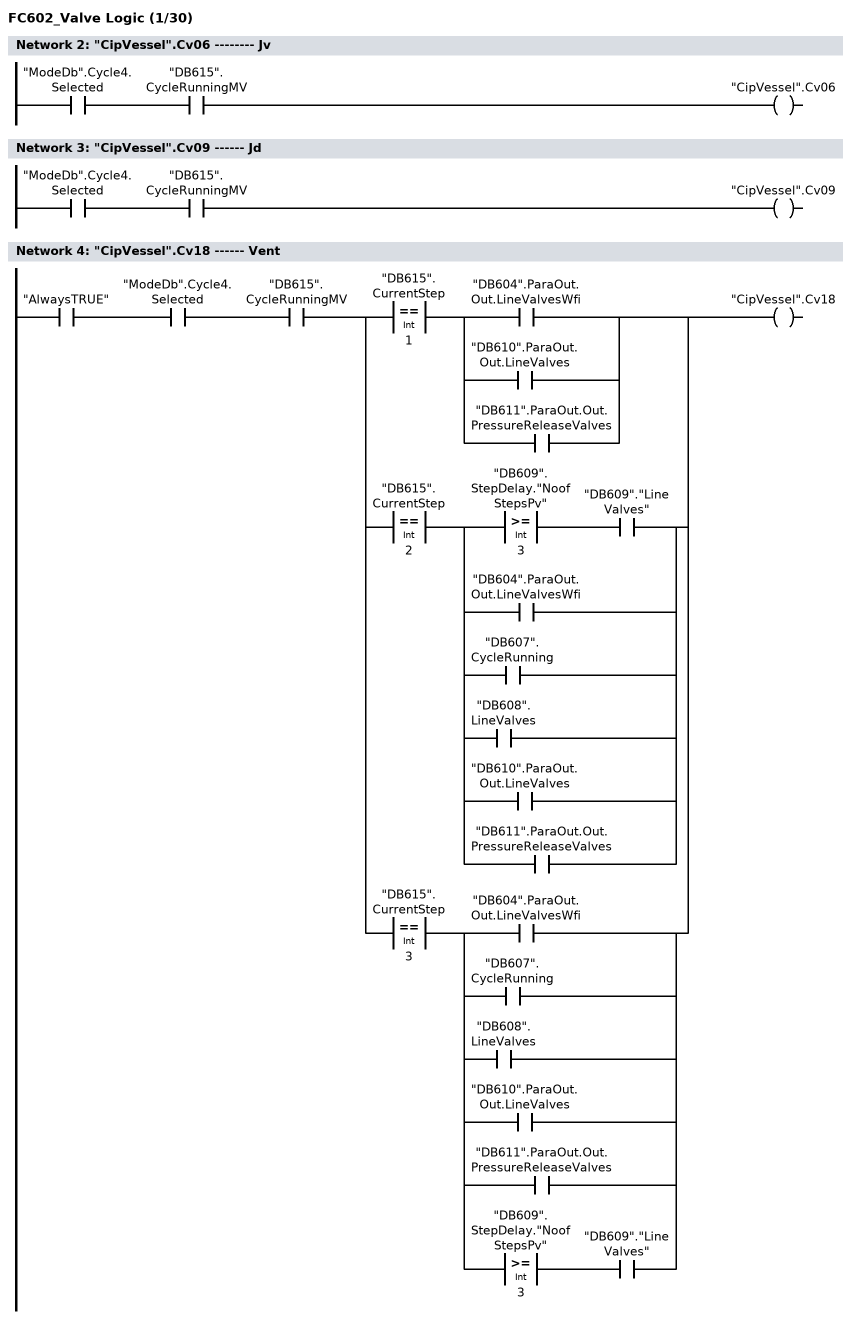
   RUNG wire#powerrail
      Contact( "ModeDb".Cycle4.Selected )
      Contact( "DB615".CycleRunningMV )
      Coil( "CipVessel".Cv06 )
   END_RUNG
   // the same network as SCL:
   "CipVessel".Cv06 := "ModeDb".Cycle4.Selected AND "DB615".CycleRunningMV;
END_REGION

REGION Network 3: "CipVessel".Cv09 ------ Jd
   RUNG wire#powerrail
      Contact( "ModeDb".Cycle4.Selected )
      Contact( "DB615".CycleRunningMV )
      Coil( "CipVessel".Cv09 )
   END_RUNG
   // the same network as SCL:
   "CipVessel".Cv09 := "ModeDb".Cycle4.Selected AND "DB615".CycleRunningMV;
END_REGION

REGION Network 4: "CipVessel".Cv18 ------ Vent
   RUNG wire#powerrail
      Contact( "AlwaysTRUE" )
      Contact( "ModeDb".Cycle4.Selected )
      Contact( "DB615".CycleRunningMV )
      wire#w1
      { S7_Templates := "SrcType := Int" } EQ_Contact(in1 := "DB615".CurrentStep, in2 := 1)
      wire#w2
      Contact( "DB604".ParaOut.Out.LineValvesWfi )
      wire#w3
      Coil( "CipVessel".Cv18 )
   END_RUNG
   RUNG wire#w2
      Contact( "DB610".ParaOut.Out.LineValves )
   END_RUNG wire#w3
   RUNG wire#w2
      Contact( "DB611".ParaOut.Out.PressureReleaseValves )
   END_RUNG wire#w3
   RUNG wire#w1
      { S7_Templates := "SrcType := Int" } EQ_Contact(in1 := "DB615".CurrentStep, in2 := 2)
      wire#w4
      { S7_Templates := "SrcType := Int" } GE_Contact(in1 := "DB609".StepDelay."Noof StepsPv", in2 := 3)
      Contact( "DB609"."Line Valves" )
   END_RUNG wire#w3
   RUNG wire#w4
      Contact( "DB604".ParaOut.Out.LineValvesWfi )
   END_RUNG wire#w3
   RUNG wire#w4
      Contact( "DB607".CycleRunning )
   END_RUNG wire#w3
   RUNG wire#w4
      Contact( "DB608".LineValves )
   END_RUNG wire#w3
   RUNG wire#w4
      Contact( "DB610".ParaOut.Out.LineValves )
   END_RUNG wire#w3
   RUNG wire#w4
      Contact( "DB611".ParaOut.Out.PressureReleaseValves )
   END_RUNG wire#w3
   RUNG wire#w1
      { S7_Templates := "SrcType := Int" } EQ_Contact(in1 := "DB615".CurrentStep, in2 := 3)
      wire#w5
      Contact( "DB604".ParaOut.Out.LineValvesWfi )
   END_RUNG wire#w3
   RUNG wire#w5
      Contact( "DB607".CycleRunning )
   END_RUNG wire#w3
   RUNG wire#w5
      Contact( "DB608".LineValves )
   END_RUNG wire#w3
   RUNG wire#w5
      Contact( "DB610".ParaOut.Out.LineValves )
   END_RUNG wire#w3
   RUNG wire#w5
      Contact( "DB611".ParaOut.Out.PressureReleaseValves )
   END_RUNG wire#w3
   RUNG wire#w5
      { S7_Templates := "SrcType := Int" } GE_Contact(in1 := "DB609".StepDelay."Noof StepsPv", in2 := 3)
      Contact( "DB609"."Line Valves" )
   END_RUNG wire#w3
   // the same network as SCL:
   "CipVessel".Cv18 := "AlwaysTRUE" AND "ModeDb".Cycle4.Selected AND "DB615".CycleRunningMV AND ((("DB615".CurrentStep = 1) AND ("DB604".ParaOut.Out.LineValvesWfi OR "DB610".ParaOut.Out.LineValves OR "DB611".ParaOut.Out.PressureReleaseValves)) OR (("DB615".CurrentStep = 2) AND ((("DB609".StepDelay."Noof StepsPv" >= 3) AND "DB609"."Line Valves") OR "DB604".ParaOut.Out.LineValvesWfi OR "DB607".CycleRunning OR "DB608".LineValves OR "DB610".ParaOut.Out.LineValves OR "DB611".ParaOut.Out.PressureReleaseValves)) OR (("DB615".CurrentStep = 3) AND ("DB604".ParaOut.Out.LineValvesWfi OR "DB607".CycleRunning OR "DB608".LineValves OR "DB610".ParaOut.Out.LineValves OR "DB611".ParaOut.Out.PressureReleaseValves OR (("DB609".StepDelay."Noof StepsPv" >= 3) AND "DB609"."Line Valves"))));
END_REGION

REGION Network 5: "CipVessel".Cv21 ------ Vent
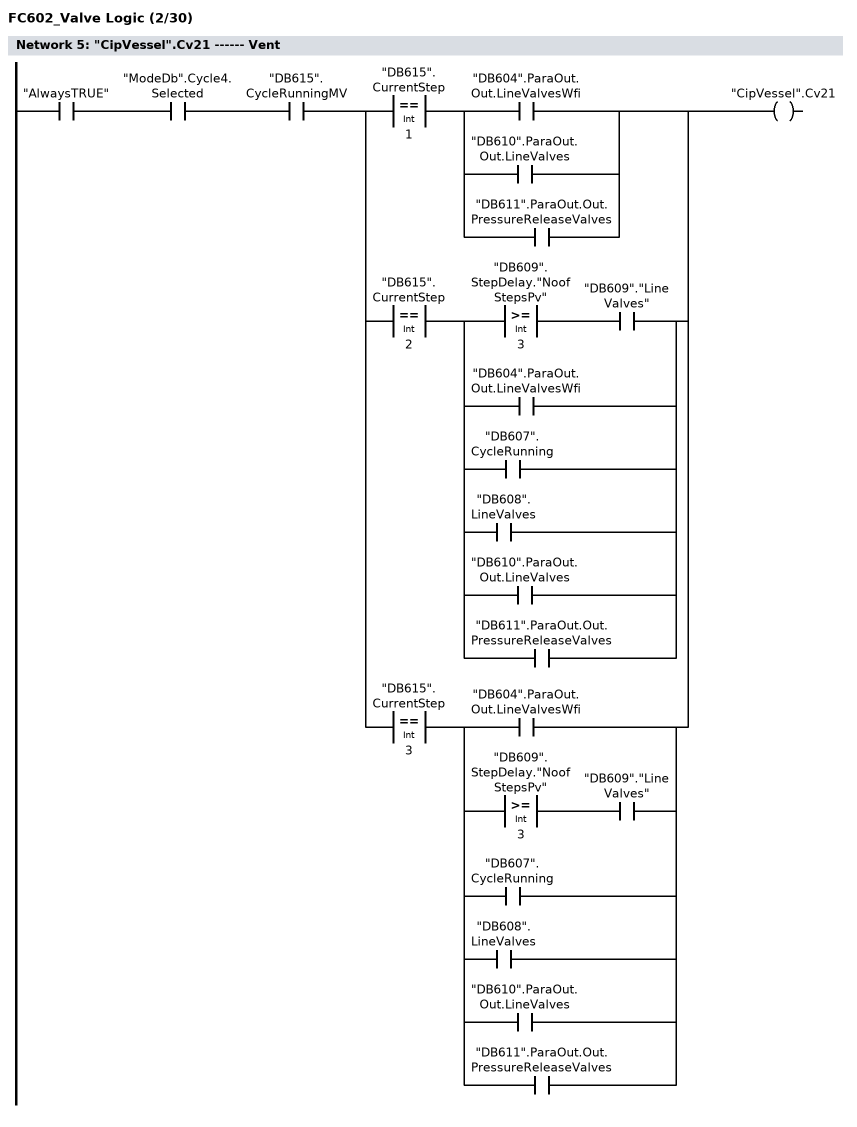
   RUNG wire#powerrail
      Contact( "AlwaysTRUE" )
      Contact( "ModeDb".Cycle4.Selected )
      Contact( "DB615".CycleRunningMV )
      wire#w1
      { S7_Templates := "SrcType := Int" } EQ_Contact(in1 := "DB615".CurrentStep, in2 := 1)
      wire#w2
      Contact( "DB604".ParaOut.Out.LineValvesWfi )
      wire#w3
      Coil( "CipVessel".Cv21 )
   END_RUNG
   RUNG wire#w2
      Contact( "DB610".ParaOut.Out.LineValves )
   END_RUNG wire#w3
   RUNG wire#w2
      Contact( "DB611".ParaOut.Out.PressureReleaseValves )
   END_RUNG wire#w3
   RUNG wire#w1
      { S7_Templates := "SrcType := Int" } EQ_Contact(in1 := "DB615".CurrentStep, in2 := 2)
      wire#w4
      { S7_Templates := "SrcType := Int" } GE_Contact(in1 := "DB609".StepDelay."Noof StepsPv", in2 := 3)
      Contact( "DB609"."Line Valves" )
   END_RUNG wire#w3
   RUNG wire#w4
      Contact( "DB604".ParaOut.Out.LineValvesWfi )
   END_RUNG wire#w3
   RUNG wire#w4
      Contact( "DB607".CycleRunning )
   END_RUNG wire#w3
   RUNG wire#w4
      Contact( "DB608".LineValves )
   END_RUNG wire#w3
   RUNG wire#w4
      Contact( "DB610".ParaOut.Out.LineValves )
   END_RUNG wire#w3
   RUNG wire#w4
      Contact( "DB611".ParaOut.Out.PressureReleaseValves )
   END_RUNG wire#w3
   RUNG wire#w1
      { S7_Templates := "SrcType := Int" } EQ_Contact(in1 := "DB615".CurrentStep, in2 := 3)
      wire#w5
      Contact( "DB604".ParaOut.Out.LineValvesWfi )
   END_RUNG wire#w3
   RUNG wire#w5
      { S7_Templates := "SrcType := Int" } GE_Contact(in1 := "DB609".StepDelay."Noof StepsPv", in2 := 3)
      Contact( "DB609"."Line Valves" )
   END_RUNG wire#w3
   RUNG wire#w5
      Contact( "DB607".CycleRunning )
   END_RUNG wire#w3
   RUNG wire#w5
      Contact( "DB608".LineValves )
   END_RUNG wire#w3
   RUNG wire#w5
      Contact( "DB610".ParaOut.Out.LineValves )
   END_RUNG wire#w3
   RUNG wire#w5
      Contact( "DB611".ParaOut.Out.PressureReleaseValves )
   END_RUNG wire#w3
   // the same network as SCL:
   "CipVessel".Cv21 := "AlwaysTRUE" AND "ModeDb".Cycle4.Selected AND "DB615".CycleRunningMV AND ((("DB615".CurrentStep = 1) AND ("DB604".ParaOut.Out.LineValvesWfi OR "DB610".ParaOut.Out.LineValves OR "DB611".ParaOut.Out.PressureReleaseValves)) OR (("DB615".CurrentStep = 2) AND ((("DB609".StepDelay."Noof StepsPv" >= 3) AND "DB609"."Line Valves") OR "DB604".ParaOut.Out.LineValvesWfi OR "DB607".CycleRunning OR "DB608".LineValves OR "DB610".ParaOut.Out.LineValves OR "DB611".ParaOut.Out.PressureReleaseValves)) OR (("DB615".CurrentStep = 3) AND ("DB604".ParaOut.Out.LineValvesWfi OR (("DB609".StepDelay."Noof StepsPv" >= 3) AND "DB609"."Line Valves") OR "DB607".CycleRunning OR "DB608".LineValves OR "DB610".ParaOut.Out.LineValves OR "DB611".ParaOut.Out.PressureReleaseValves)));
END_REGION

REGION Network 6: "CipVessel".Cv02 ------ Wfi
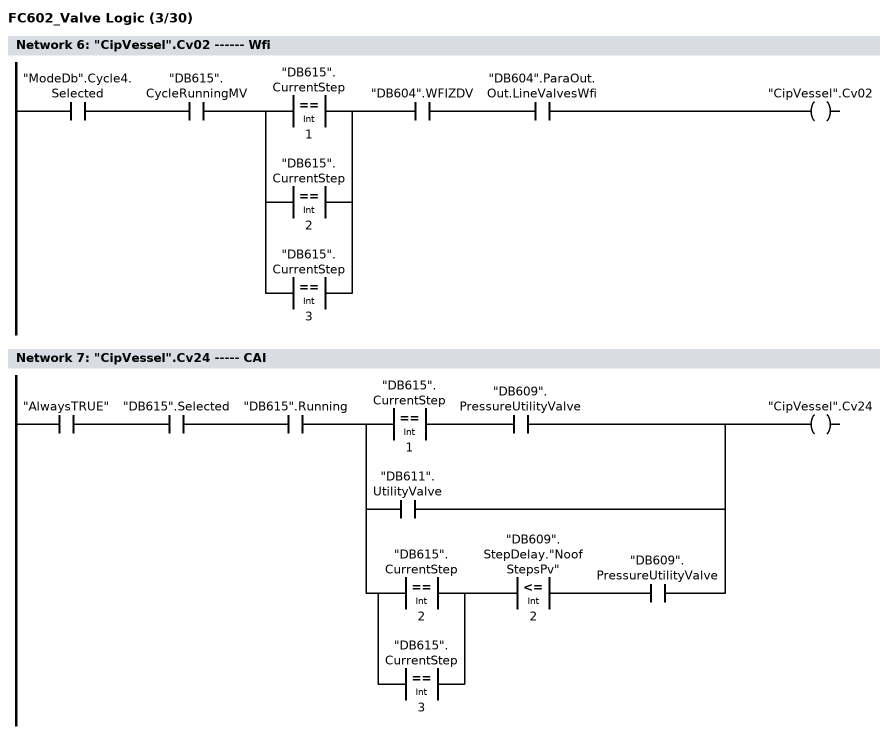
   RUNG wire#powerrail
      Contact( "ModeDb".Cycle4.Selected )
      Contact( "DB615".CycleRunningMV )
      wire#w1
      { S7_Templates := "SrcType := Int" } EQ_Contact(in1 := "DB615".CurrentStep, in2 := 1)
      wire#w2
      Contact( "DB604".WFIZDV )
      Contact( "DB604".ParaOut.Out.LineValvesWfi )
      Coil( "CipVessel".Cv02 )
   END_RUNG
   RUNG wire#w1
      { S7_Templates := "SrcType := Int" } EQ_Contact(in1 := "DB615".CurrentStep, in2 := 2)
   END_RUNG wire#w2
   RUNG wire#w1
      { S7_Templates := "SrcType := Int" } EQ_Contact(in1 := "DB615".CurrentStep, in2 := 3)
   END_RUNG wire#w2
   // the same network as SCL:
   "CipVessel".Cv02 := "ModeDb".Cycle4.Selected AND "DB615".CycleRunningMV AND (("DB615".CurrentStep = 1) OR ("DB615".CurrentStep = 2) OR ("DB615".CurrentStep = 3)) AND "DB604".WFIZDV AND "DB604".ParaOut.Out.LineValvesWfi;
END_REGION

REGION Network 7: "CipVessel".Cv24 ----- CAI
   RUNG wire#powerrail
      Contact( "AlwaysTRUE" )
      Contact( "DB615".Selected )
      Contact( "DB615".Running )
      wire#w1
      { S7_Templates := "SrcType := Int" } EQ_Contact(in1 := "DB615".CurrentStep, in2 := 1)
      Contact( "DB609".PressureUtilityValve )
      wire#w2
      Coil( "CipVessel".Cv24 )
   END_RUNG
   RUNG wire#w1
      Contact( "DB611".UtilityValve )
   END_RUNG wire#w2
   RUNG wire#w1
      { S7_Templates := "SrcType := Int" } EQ_Contact(in1 := "DB615".CurrentStep, in2 := 2)
      wire#w3
      { S7_Templates := "SrcType := Int" } LE_Contact(in1 := "DB609".StepDelay."Noof StepsPv", in2 := 2)
      Contact( "DB609".PressureUtilityValve )
   END_RUNG wire#w2
   RUNG wire#w1
      { S7_Templates := "SrcType := Int" } EQ_Contact(in1 := "DB615".CurrentStep, in2 := 3)
   END_RUNG wire#w3
   // the same network as SCL:
   "CipVessel".Cv24 := "AlwaysTRUE" AND "DB615".Selected AND "DB615".Running AND ((("DB615".CurrentStep = 1) AND "DB609".PressureUtilityValve) OR "DB611".UtilityValve OR ((("DB615".CurrentStep = 2) OR ("DB615".CurrentStep = 3)) AND ("DB609".StepDelay."Noof StepsPv" <= 2) AND "DB609".PressureUtilityValve));
END_REGION

REGION Network 8: "CipVessel".Cv17 ----- N2B
